(* PLC project 1m8QV2026年3月28日 - 信号稳定延长 - 10ms - 副本.project, CODESYS CODESYS V3.5 SP18 *)
(* stored: creationDateTime 2026-06-03T09:30:15.46669, modificationDateTime 2026-06-01T11:36:08.9259729 *)

(* ============================================================================== DUT: AxisCrtlStruct 作用: 单轴“控制意图”数据结构；每轴各有一份 Local（本控）与 Remote（远控） 使用者: *_Ctrl_FB（读 sCtrl/sLocal）、*_ctrl_1、SecurityCheck、Modbus_Slave ============================================================================== *)
TYPE AxisCrtlStruct : STRUCT
  iMode : INT;  (* 当前请求模式，取值见 MODES 枚举 *)
  rPosCmd : REAL;  (* 位置命令 (deg)，位置/程引模式目标 *)
  rVelCmd : REAL;  (* 速度命令 (deg/s)，速度模式目标 *)
  rPIDCmdVel : LREAL;  (* PID 输出的速度指令（内部，写 CANopen 目标速度前） *)
  rPIDCmdPos : LREAL;  (* PID 目标位置（内部） *)
  bPIDEnable : BOOL;  (* 位置环 PID 使能 *)
  bStartAutoTrack : BOOL;  (* 自跟踪使能：TRUE 时用 rChanU 误差驱动 *)
  rChanU : REAL;  (* 跟踪接收机误差电压（自跟踪通道） *)
  rP : REAL := 1.0;  (* PID 比例系数（正常指向） *)
  rI : REAL := 0;  (* PID 积分系数 *)
  rD : REAL := 0;  (* PID 微分系数 *)
  rPIDThre : INT := 1;  (* 积分开启的位置误差阈值 *)
  rP_AutoTrack : REAL := 3.0;  (* 自跟踪 P *)
  rI_AutoTrack : REAL := 0.02;  (* 自跟踪 I *)
  rAcceleration : REAL := 3;  (* 加速度 (deg/s²)，写 diTargetAcc 前换算 *)
  rDeceleration : REAL := 3;  (* 减速度 (deg/s²) *)
  rJogVel : LREAL := 2;  (* 点动速度 *)
  Pos_Vel : REAL := 4;  (* 位置模式最大趋近速度 (deg/s) *)
  rPos_Limit : LREAL;  (* 位置限位（备用） *)
  rVel_Limit : LREAL := 3;  (* 速度限幅 (deg/s) *)
  rSoft_limit_Postive : REAL;  (* 软限位正限 (deg) *)
  rSoft_limit_Negative : REAL;  (* 软限位负限 (deg) *)
  rLimitionNegative : LREAL;  (* 硬限位负（备用） *)
  rLimitionPositive : LREAL;  (* 硬限位正（备用） *)
END_STRUCT;
END_TYPE

(* ============================================================================== DUT: AxisStatus 作用: 单轴运行状态（由 *_ctrl_1 根据 CANopen 状态字/逻辑填写） 使用者: *_Ctrl_FB（判断 Disabled/Moving）、Modbus 上报、HMI ============================================================================== *)
TYPE AxisStatus : STRUCT
  Valid : BOOL;  (* 轴数据有效（SoftMotion 风格字段，部分逻辑未用） *)
  Busy : BOOL;  (* 轴忙 *)
  Error : BOOL;  (* 有故障（常映射 GVL.bXxxStsBit3） *)
  ErrorID : UINT;  (* 故障码（常映射 eXxxErrorcode） *)
  ErrorStop : BOOL;  (* 故障停机中 *)
  Disabled : BOOL;  (* 伺服未使能/下电状态 *)
  Stopping : BOOL;  (* 正在停止 *)
  Homing : BOOL;  (* 回零中 *)
  Standstill : BOOL;  (* 静止 Standstill *)
  DiscreteMotion : BOOL;  (* 离散运动 *)
  ContinuousMotion : BOOL;  (* 连续运动 *)
  bServo_Enable : BOOL;  (* 伺服已使能（本工程：StsBit0/1/2 均为真） *)
  bBrake : BOOL;  (* 抱闸抱紧（与使能相反） *)
  Moving : BOOL;  (* 是否在运动（ctrl_1 根据速度判断 bStop_x） *)
END_STRUCT;
END_TYPE

(* ============================================================================== DUT: AxisVisible 作用: 本控/HMI 显示与操作相关状态（可视化、按钮灯） 使用者: 可视化或本控面板逻辑（部分工程可能未全部接线） ============================================================================== *)
TYPE AxisVisible : STRUCT
  bJog_Forward : BOOL := FALSE;
  bJog_Backward : BOOL := FALSE;
  bVel_Run : BOOL := FALSE;
  bPos_Run : BOOL := FALSE;
  bEnable : BOOL;  (* 使能指示灯 *)
  bUnable : BOOL;  (* 下使能指示灯 *)
  bLocalCtrl : BOOL;  (* 本控指示灯 *)
  bRemoteCtrl : BOOL;  (* 远控指示灯 *)
  bStop : BOOL;  (* 停止指示灯 *)
  bmoveLight : BOOL;
  bErrLight : BOOL;  (* 报错提示灯 *)
  rLocalPosCmd : REAL;  (* 本控位置命令 *)
  rLocalVelCmd : REAL;  (* 本控速度命令 *)
END_STRUCT;
END_TYPE

(* values of MODES: powerOff: 下电：断开驱动使能、清零控制字; powerOn: 上电：按步序置位 bCtrlBit，准备伺服; positionMode: 位置模式：位置环/指向，远控指向常用; velocityMode: 手动速度模式：直接写目标速度; programBootMode: 程序引导/程引模式：按时间插值位置（RealTimePosCal）; reset: 轴错误复位（配合 GVL.bError_Reset）; halt: 停止：减速停机; stop: 挂机/保持停止; jog: 退限位/点动类模式; edge: 边沿相关模式（工程内扩展用）; test1: 测试/多项式系数下发等扩展模式 *)

(* ============================================================================== DUT: MODES 作用: 三轴运动控制状态机使用的模式枚举（El_Ctrl_FB 等 CASE iMode OF） 用法: sCtrl.iMode / sLocal.iMode 与 MODES.xxx 比较 注意: 数值 5 未使用；test1(11) 用于多项式等特殊调试 ============================================================================== *)
{attribute 'qualified_only'}
{attribute 'strict'}
TYPE MODES : (powerOff := 0, powerOn := 1, positionMode := 2, velocityMode := 3, programBootMode := 4, reset := 6, halt := 7, stop := 8, jog := 9, edge := 10, test1 := 11);
END_TYPE

TYPE Word2Bit : UNION
  Apart_Word : WORD;  (* 整字视图（如 AGC 原始 WORD） *)
  Apart_Byte : ARRAY[1..2] OF BYTE;  (* 按字节拆分，[1][2] 与串口 recBuf 逐字节对接 *)
  Apart_Real : REAL;  (* 按 32 位实数解释（本 UNION 仅 16 位，慎用） *)
  Apart_Int : INT;  (* 有符号整数视图（如 Ua/Ue 误差电压 raw） *)
END_UNION;
END_TYPE

TYPE Dword2Bit : UNION
  Apart_Dword : DWORD;  (* 32 位整字 *)
  Apart_Word : ARRAY[1..2] OF WORD;  (* 拆成两个 16 位寄存器（与 Modbus WORD 对接时常用） *)
  Apart_Byte : ARRAY[1..4] OF BYTE;  (* 4 字节，串口按字节填充 *)
  Apart_Real : REAL;  (* 32 位浮点视图 *)
  Apart_Int : INT;  (* 32 位有符号整数（部分帧解析用 INT） *)
END_UNION;
END_TYPE

TYPE float2bit : UNION
  Apart_ulint : ULINT;  (* 64 位无符号时间戳等 *)
  Apart_dword : ARRAY[1..2] OF DWORD;  (* 两个双字；位置常用 dword[1] 装 DINT *)
  Apart_word : ARRAY[1..4] OF WORD;  (* 四个 Modbus 保持寄存器字 *)
  Apart_byte : ARRAY[1..8] OF BYTE;  (* 8 字节逐字节访问 *)
  Apart_real : ARRAY[1..2] OF REAL;  (* 两个 REAL 视图 *)
  Apart_int : ARRAY[1..4] OF INT;  (* 四个 INT 视图 *)
END_UNION;
END_TYPE

TYPE UnionLREAL_WORD : UNION
  lrealValue : LREAL;  (* 程序内使用的双精度浮点值 *)
  words : ARRAY[1..4] OF WORD;  (* Modbus 4 寄存器拼装/拆分 *)
END_UNION;
END_TYPE

TYPE Time2Word : UNION
  uliData : ULINT;  (* 64 位时间（如 ns/ms 打包，视使用处换算） *)
  wWords : ARRAY[1..4] OF WORD;  (* 与 4 个寄存器对应 *)
  lrReal : LREAL;  (* 双精度时间或系数视图 *)
  arReal : ARRAY[0..1] OF REAL;  (* 两个单精度视图（高低段等） *)
END_UNION;
END_TYPE

PROGRAM PLC_PRG
  VAR
    a : DINT;
    b : REAL;
  END_VAR

                    a := REAL_TO_DINT(b * 524288 / 360);
                  
END_PROGRAM

PROGRAM TimeCase
  VAR
    Triger AT %IX0.0 : BOOL;
    Feed AT %QX0.0 : BOOL;
  END_VAR
  VAR
    stUTC_Timestamp : SYSTIME;
    stSYS_Timestamp : ULINT;
    stGNSS_Timestap : ULINT;
    Result : RTS_IEC_RESULT;
    Uptriger : Standard.R_TRIG;
    TON_F : TON;
    dDelPTime : DINT;
    max_DelPTime : DINT := 0;
    min_DelPTime : DINT := -999999;
    iCount : INT;
    dtNow : DT;
    dtGNSS : DT;
    dtLastGNSS : ULINT;
    iDiffETime : DINT;
    DelPTime : DINT;
  END_VAR

                    //计算时间误差序列
Result := SysTimeRtcHighResGet(stUTC_Timestamp);        
stSYS_Timestamp := TO_ULINT(stUTC_Timestamp);           // ULINT，获取本地时间
dtNow := TO_DT(stUTC_Timestamp / 1000); 		        // 转换为DATE_AND_TIME类型

Uptriger(CLK:=Triger);                                  //检测PPS上升沿
IF Uptriger.Q THEN                                      //上升沿触发后，GPRMC解析，DO0上升沿输出（电平24V）
	Feed:=TRUE;	
	dtGNSS := TO_DT(GVL.stGNSS_Timestap / 1000); 	    // 拿到串口时间数据			                                     
	iDiffETime:=ULINT_TO_DINT(GVL.stGNSS_Timestap-dtLastGNSS);  
	dtLastGNSS:=GVL.stGNSS_Timestap;                    //缓存上一周期时间戳（ms)  
	dDelPTime:=ULINT_TO_DINT(GVL.stGNSS_Timestap - stSYS_Timestamp);       //计算误差	              
	IF iDiffETime = 1000 THEN                           //确保时间更新步进1S
		IF dDelPTime < 0 THEN                           //更新最小值
			IF dDelPTime < min_DelPTime THEN
				min_DelPTime:=dDelPTime;
				DelPTime:=min_DelPTime;                 
			END_IF		
		ELSE                                            //更新最大值
			IF dDelPTime > max_DelPTime THEN
				max_DelPTime:=dDelPTime;
				DelPTime:=max_DelPTime;
			END_IF
		END_IF	
	END_IF				    						
	iCount:=iCount+1;
	IF iCount >= 60 THEN                                //一分钟校一次时间
		GVL.dDelTime:=DelPTime;
		max_DelPTime:=0;
		min_DelPTime:=0;	
		iCount:=0;
	END_IF
	
END_IF
TON_F(IN:=Feed, PT:=T#100MS, Q=>,ET=>);                 //脉宽200ms（测试时延，为了在示波器看波形）
IF TON_F.Q THEN
	Feed:=FALSE;		
END_IF
                  
END_PROGRAM

FUNCTION_BLOCK PID
  VAR_INPUT
    rTarget : REAL;  (* 目标位置 (deg) *)
    rFeedback : REAL;  (* 实际位置反馈 (deg) *)
    rPosLimPositive : LREAL;  (* 软限位正限 (deg)，超出则输出清零 *)
    rPosLimNegative : LREAL;  (* 软限位负限 (deg) *)
    rKp : REAL;  (* 比例系数 *)
    rKi : REAL;  (* 积分系数 *)
    rKd : REAL;  (* 微分系数（当前逻辑未实际使用） *)
    iThreshold : INT;  (* 积分开启阈值 (deg)；-1 = 始终开积分 *)
    bPIDEnable : BOOL;  (* PID 使能，FALSE 时各项清零 *)
    rVelLim : LREAL;  (* 输出速度限幅 (deg/s) *)
  END_VAR
  VAR_OUTPUT
    rPIDOutput : LREAL;  (* PID 输出速度 (deg/s)，写到 diXxTargetVel 前换算 *)
    rPIDtrace : LREAL;  (* 调试/显示用，与 rPIDOutput 相同 *)
  END_VAR
  VAR
    rLastError : LREAL;  (* 上一拍误差（当前版本未使用微分，保留备用） *)
    rErrorNow : LREAL;  (* 当前误差 = rTarget - rFeedback *)
    rIntegralNew : LREAL;  (* 积分累计量 *)
    rDerivativeNew : LREAL;  (* 微分项（未使用） *)
    rDelta : LREAL;  (* 备用 *)
    rProportionNew : LREAL;  (* 比例项 = rErrorNow *)
  END_VAR

                    
(*==============================================================================
  FB: PID（位置环速度输出 PID）
  任务: Canopen 10ms（由 *_Ctrl_FB 调用）
  作用: 输入目标位置与实际位置，输出速度指令（deg/s）
  算法: 比例 + 条件积分（误差小于阈值才累积），无微分
  使用者: El_Ctrl_FB / Az_Ctrl_FB / Ti_Ctrl_FB 中的 VelPID_1/2/3
==============================================================================*)

// ----- 段：PID 使能入口 -----
IF (bPIDEnable>0) THEN //如果PID使能
	IF rTarget=rFeedback THEN
		rPIDOutput:=0;	               // 目标=反馈，输出为 0
	ELSE
	
		rErrorNow:=rTarget-rFeedback;  //计算当前误差 en
		rProportionNew:=rErrorNow;     //比例项

		// ----- 段：条件积分（仅在软限位内、误差小于阈值时才累积）-----
		IF rFeedback>rPosLimNegative AND rFeedback<rPosLimPositive THEN //若在软限位之内，工作时开启积分项
			IF (ABS(rTarget-rFeedback)<iThreshold) THEN//位置差小于积分阈值
				rIntegralNew:= rIntegralNew+rErrorNow; //积分项
			ELSE
				rIntegralNew:=0;
			END_IF;
		ELSE //不在软限位范围内,则积分项为0
			rIntegralNew:=0;
		END_IF

		// ----- 段：PID 求和输出 -----
		rPIDOutPut:=rKp*rProportionNew+rKi*rIntegralNew;
		rPIDtrace:=rKp*rProportionNew+rKi*rIntegralNew;

		// ----- 段：速度限幅（双向） -----
		IF rPIDOutput<(-rVelLim) THEN
			rPIDOutput:=-rVelLim;
		ELSIF rPIDOutput>rVelLim THEN
			rPIDOutput:=rVelLim;
		END_IF
		
		// ----- 段：超软限位时强制输出清零，防止继续向限位方向运动 -----
		IF rFeedback>rPosLimPositive AND rPIDOutput>0 THEN 
			rPIDOutput:=0;
		END_IF
		IF rFeedback<rPosLimNegative AND rPIDOutput<0 THEN
			rPIDOutput:=0;
		END_IF
		
		rLastError:=rErrorNow;//将当前误差赋值给上一次误差
		
	END_IF
ELSE//非使能清零PID各项
	rProportionNew:=0.0;
	rIntegralNew:=0.0;
	rPIDOutput:=0.0;
END_IF





                  
END_FUNCTION_BLOCK

PROGRAM TimeAdd
  VAR
    icount : INT;
    iSecondLast : INT;
  END_VAR

                    
(*==============================================================================
  PRG: TimeAdd（GNSS 秒跳变监测 / 毫秒插值计数）
  任务: Canopen 10ms
  作用:
    - 监测 GPRMC_1.iSecond 是否更新；未更新则 icount 每 10ms +1
    - RealTimePosCal 使用: GVL.dRealTime := GVL.stGNSS_Timestap + 10 * TimeAdd.icount
      即在两次 GNSS 报文之间用 10ms 步进“补时”，保证程引插值时间连续
  说明:
    icount>2000 时清零（约 20s 无新秒则复位，防止溢出跑飞）
==============================================================================*)
// 监测时统串口状态，时间插值
IF iSecondLast <> GPRMC_1.iSecond THEN
	icount := 0;
ELSE
	icount := icount + 1;
END_IF
iSecondLast := GPRMC_1.iSecond;

IF icount > 2000 THEN
	icount := 0;
END_IF
                  
END_PROGRAM

PROGRAM GPRMC
  VAR
    com_init : gcan.FB_Com_Init;  (* gcan.FB_Com_Init为串口初始化功能块，可设定串口端口号，串口波特率等参数 *)
    com_read : gcan.FB_Com_Read;  (* gcan.FB_Com_Read为串口接收功能块，用于通过接收串口发送给PLC的数据 *)
    com_write : gcan.FB_Com_Write;  (* gcan.FB_Com_Write为串口发送功能块，用于发送串口数据 *)
    m_uiError : UINT;  (* 用于承接功能块中报错引脚错误信息的变量 *)
    m_out : BOOL;  (* 用于承接功能块中完成标志引脚数据的变量 *)
    isFirst : BOOL := TRUE;  (* 用于判断初始化只执行一次的逻辑 *)
    mPort : BYTE;  (* 程序中用作设定串口端口号 *)
    recSize : UINT;  (* 接收数据长度，单位：字节 *)
    recBuf : ARRAY[0..100] OF BYTE;  (* 用于存放接收到的串口数据的数组 *)
    sum_i : INT;
    checksum : BYTE;
    iYear : INT;
    iMonth : INT;
    iDay : INT;
    iHour : INT;
    iMinute : INT;
    iSecond : INT;
    strDateTimeNow : STRING;
    gnssTimestamp : ULINT;
    high4 : BYTE;
    low4 : BYTE;
  END_VAR

                    ////////////////////////////////////////////////////////////////////////////////////////
//串口接收GPRMC报文解析
//日期：2024/08/25
//版本：V1.1
/////////////////////////////////////////////////////////////////////////////////////////

mPort:=1;								//串口端口号设定，GCAN-PLC-400、GCAN-PLC-510、GCAN-PLC-511，1为232，2为485
										//GCAN-PLC-324、GCAN-PLC-326，1为第一路485，2为第2路485
IF isFirst THEN
	com_init(							//串口初始化功能块
	EN_IN:=TRUE,						//串口初始化功能块使能
	xEnable:=TRUE,						//串口功能使能
	bPort:=mPort,						//串口端口号设定
	uiBaudrate:=115200,					//串口波特率设定
	bParity:=0,							//串口奇偶校验设定，0为无校验，1为奇校验，2为偶检验
	bDatabits:=8,						//数据位设定
	bStopbits:=1,						//停止位设定
	EN_OUT=>m_out,						//串口初始化功能块执行完成标志位
	uiError=>m_uiError);				//串口初始化功能块执行错误信息
	isfirst:=FALSE;						//执行一次初始化后关闭IF的条件使其之后进入ELSE程序段运行

ELSE
	
		com_read(						//串口读取功能块
		EN_in:=TRUE,					//读取功能块使能，为TRUE执行读取
		bPort:=mPort,					//串口端口号设定
		p_brxdata:=ADR(recBuf),			//读取到的串口数据引脚为指针类型，使用ADR()指向自建数组将数据存放到数组中
		uiMaxsize:=100,					//设定最大读取长度
		EN_out=>m_out,					//串口读取功能块执行完成标志位******功能块执行完成不代表接收完成********
		uiRecSize=>recSize,				//串口接收数据长度，单位：字节，大于0时说明接收到数据可用于判断是否接收
		uierror=>m_uierror);			//串口读取功能块执行错误信息
										//从数组recBuf里取数据，解析出年、月、日、时、分、秒
		//有效判定(A)+和校验(hh),前 4bit和后 4bit的 16 进制数分别以 ASCII 码表示(0~9,A~F)，高位在前。
		IF 	recBuf[17] = 65 THEN
(*			checksum := 16#00;
			FOR sum_i:=1 TO 74 BY 1 DO
				checksum:= checksum XOR recBuf[sum_i];
			END_FOR
			high4 := (SHR(checksum, 4) AND 16#0F)+16#30;
			low4 := (checksum AND 16#0F)+16#30;
			IF recBuf[76]= high4 AND recBuf[77]= low4 THEN 
*)			IF recBuf[60] = 44 THEN // 航向角 x.x
				iYear:=BYTE_TO_INT(recBuf[65]-48)*10+BYTE_TO_INT(recBuf[66]-48)+2000;
				iMonth:=BYTE_TO_INT(recBuf[63]-48)*10+BYTE_TO_INT(recBuf[64]-48);
				iDay:=BYTE_TO_INT(recBuf[61]-48)*10+BYTE_TO_INT(recBuf[62]-48);
				iHour:=BYTE_TO_INT(recBuf[7]-48)*10+BYTE_TO_INT(recBuf[8]-48)+8;
				iMinute:=BYTE_TO_INT(recBuf[9]-48)*10+BYTE_TO_INT(recBuf[10]-48);
				iSecond:=BYTE_TO_INT(recBuf[11]-48)*10+BYTE_TO_INT(recBuf[12]-48);
			END_IF
			IF recBuf[61] = 44 THEN // 航向角 xx.x
				iYear:=BYTE_TO_INT(recBuf[66]-48)*10+BYTE_TO_INT(recBuf[67]-48)+2000;
				iMonth:=BYTE_TO_INT(recBuf[64]-48)*10+BYTE_TO_INT(recBuf[65]-48);
				iDay:=BYTE_TO_INT(recBuf[62]-48)*10+BYTE_TO_INT(recBuf[63]-48);
				iHour:=BYTE_TO_INT(recBuf[7]-48)*10+BYTE_TO_INT(recBuf[8]-48)+8;
				iMinute:=BYTE_TO_INT(recBuf[9]-48)*10+BYTE_TO_INT(recBuf[10]-48);
				iSecond:=BYTE_TO_INT(recBuf[11]-48)*10+BYTE_TO_INT(recBuf[12]-48);
			END_IF
			IF recBuf[62] = 44 THEN // 航向角 xxx.x
				iYear:=BYTE_TO_INT(recBuf[67]-48)*10+BYTE_TO_INT(recBuf[68]-48)+2000;
				iMonth:=BYTE_TO_INT(recBuf[65]-48)*10+BYTE_TO_INT(recBuf[66]-48);
				iDay:=BYTE_TO_INT(recBuf[63]-48)*10+BYTE_TO_INT(recBuf[64]-48);
				iHour:=BYTE_TO_INT(recBuf[7]-48)*10+BYTE_TO_INT(recBuf[8]-48)+8;
				iMinute:=BYTE_TO_INT(recBuf[9]-48)*10+BYTE_TO_INT(recBuf[10]-48);
				iSecond:=BYTE_TO_INT(recBuf[11]-48)*10+BYTE_TO_INT(recBuf[12]-48);
			END_IF
				// 计算时间戳		
				strDateTimeNow := CONCAT(STR1 := 'DT#', STR2 := INT_TO_STRING(iYear));
				strDateTimeNow := CONCAT(STR1 := strDateTimeNow, STR2 := '-');
				strDateTimeNow := CONCAT(STR1 := strDateTimeNow, STR2 := INT_TO_STRING(iMonth));
				strDateTimeNow := CONCAT(STR1 := strDateTimeNow, STR2 := '-');
				strDateTimeNow := CONCAT(STR1 := strDateTimeNow, STR2 := INT_TO_STRING(iDay));
				strDateTimeNow := CONCAT(STR1 := strDateTimeNow, STR2 := '-');
				strDateTimeNow := CONCAT(STR1 := strDateTimeNow, STR2 := INT_TO_STRING(iHour));
				strDateTimeNow := CONCAT(STR1 := strDateTimeNow, STR2 := ':');
				strDateTimeNow := CONCAT(STR1 := strDateTimeNow, STR2 := INT_TO_STRING(iMinute));
				strDateTimeNow := CONCAT(STR1 := strDateTimeNow, STR2 := ':');
				strDateTimeNow := CONCAT(STR1 := strDateTimeNow, STR2 := INT_TO_STRING(iSecond));
				gnssTimestamp := DT_TO_ULINT(TO_DT(strDateTimeNow)) * 1000;
				GVL.stGNSS_Timestap := gnssTimestamp;
			//END_IF
		END_IF
					


(*	IF recsize>0 THEN					//如果接收到串口数据
		
		com_write(						//串口发送功能块
		EN_IN:=TRUE,					//串口发送功能块使能，发送机制：当使能为TRUE时，PLC程序每周期运行到此处就执行一次发送
		bPort:=mPort,					//串口端口号设定
		p_bTxdata:=ADR(recbuf),			//将接收存放到数组中的数据发送出去******若发送其它数据，自建另一数组用于存放发送数据即可
		uiTxsize:=recsize,				//发送长度为接收到的数据长度******若发送其它长度，自行填写所需长度即可
		EN_OUT=>m_out,					//串口发送功能块执行完成标志位
		uierror=>m_uierror);			//串口发送功能块执行错误信息
			
	END_IF
*)	
END_IF
                  
END_PROGRAM

PROGRAM RealTimePosCal
  VAR
    dtReal : DT;
    sRealTime : STRING;
    btestTimeInit : BOOL;
    AzCubicInter : threesimple2_1;  (* 方位三次样条插值 *)
    ElCubicInter : threesimple2_1;  (* 俯仰三次样条插值 *)
    iErrcode : INT;
    rInterAzPos : REAL;  (* 方位轴插值位置 *)
    rInterElPos : REAL;  (* 俯仰轴插值位置 *)
    rInterAzPostest : REAL;  (* 方位轴插值位置 *)
    rInterElPostest : REAL;  (* 俯仰轴插值位置 *)
    rPolyAzPos : REAL;  (* 方位轴多项式位置 *)
    rPolyElPos : REAL;  (* 俯仰轴多项式位置 *)
    AzPoly : Get_AZ;
    ElPoly : Get_AZ_1;
    dRTime : ULINT;  (* 上位机外部时间 单位ns Unix时间戳，起点是1970-1-1 0:0:0 *)
    dLastRTime : ULINT;
    icount : INT;
  END_VAR

                    
(*==============================================================================
  PRG: RealTimePosCal（程引实时位置计算）
  任务: Canopen 10ms
  作用:
    1. 合成 GVL.dRealTime（毫秒时间轴，供插值用 xt）
    2. 双轴程引(mode4)时，按时间对 Modbus 轨道表做三次样条插值
    3. 输出 rInterAzPos / rInterElPos → *_ctrl_1 合成 rPIDCmdPos
  时间源（GVL.bTimeSwich）:
    FALSE — GNSS: stGNSS_Timestap + 10×TimeAdd.icount
    TRUE  — 上位机 UTC: Modbus_Slave.UTC_New + 8h + 10×本地 icount
  插值输入:
    X = Modbus_Slave.aUTC_TIME[1..10]（时间结点，相对首点归一化）
    Y = Modbus_Slave.aPosCmd_1/2（俯仰/方位角度结点）
    xt = dRealTime - 8×3600×1000（转为与轨道表一致的 UTC 毫秒）
==============================================================================*)

// =============================================================================
// 段 1: 合成 GVL.dRealTime（全局毫秒时钟）
// =============================================================================

//直接从上位机拿数（UTC_New 一般为 UTC 毫秒，+8h 对齐北京时）
dRTime := modbus_slave.UTC_New + 8 * 3600 * 1000;
IF dRTime <> dLastRTime THEN
	icount := 0;
ELSE 
	icount := icount + 1;
END_IF
dLastRTime:=dRTime;

IF not GVL.bTimeSwich THEN
	GVL.dRealTime:=GVL.stGNSS_Timestap + 10*timeadd.icount;   // GNSS + 插值
ELSE
	GVL.dRealTime:=dRTime + 10*icount;                        // 上位机 UTC + 插值
END_IF
IF icount > 5000 THEN
	icount := 0;
END_IF
(*
GVL.dRealTime:=GVL.stGNSS_Timestap + 10*timeadd.icount;
*)
dtReal := TO_DT(GVL.dRealTime / 1000);
sRealTime := TO_STRING(dtReal);

// =============================================================================
// 段 2: 双轴均为程引 mode4 时 — 三次样条插值求当前俯仰/方位
// xt 减去 8×3600×1000 与轨道表 aUTC_TIME 时间基准对齐
// =============================================================================
IF Axis1Remote.iMode=4 AND Axis2Remote.iMode=4 THEN//若PTP时间锁定 且时间模式为PTP时间
		//三次样条插值

		//GVL.dRealTime:= TimeCase.stSYS_Timestamp + GVL.dDelTime + 1000 + 56; // 矫正后的时间 单位毫秒
		IF NOT GVL.bTimeSwich THEN
			GVL.dRealTime:=GVL.stGNSS_Timestap + 10*timeadd.icount;
		ELSE
			GVL.dRealTime:=dRTime + 10*icount;
		END_IF
		AzCubicInter(XModbusUL:=Modbus_Slave.aUTC_TIME,YModbus:=Modbus_Slave.aPosCmd_2,y0:=0,yn:=0,xt:=(ULINT_TO_LREAL(GVL.dRealTime) - 8 * 3600 *1000),sout=>rInterAzPos,ErrCode=>iErrcode);
		ElCubicInter(XModbusUL:=Modbus_Slave.aUTC_TIME,YModbus:=Modbus_Slave.aPosCmd_1,y0:=0,yn:=0,xt:=(ULINT_TO_LREAL(GVL.dRealTime) - 8 * 3600 *1000),sout=>rInterElPos,ErrCode=>iErrcode);
		IF iErrcode>0 THEN //模块内错误代码清0 外部维持
			Error_code:=iErrcode;
		END_IF
END_IF

(* 段 3: 多项式拟合程引（Get_AZ / Get_AZ_1）整段已注释，当前未使用
   若启用: rInterAzPos = -rPolyAzPos, rInterElPos = rPolyElPos + 90
*)

                  
END_PROGRAM

PROGRAM Modbus_Slave
  VAR
    modbusData AT %MW0 : ARRAY[0..654] OF WORD;  (* HR 保持寄存器，CODESYS 地址 %MW0 起 *)
    modbusInputRegs AT %MW660 : ARRAY[0..79] OF WORD;  (* IR 输入寄存器，%MW660 起 *)
  END_VAR
  VAR
    modTcpSlaveInit : gcan.FB_ModbusTCP_Slave_Init;  (* ----- Modbus TCP 协议栈 ----- *)
    modTcpSlaveCtrl : gcan.FB_ModbusTCP_Slave_Ctrl;
    eout : BOOL;
    iSocket : INT;
    uiErr : UINT;
    isInit : BOOL;
    arClient : ARRAY[0..10] OF INT;
    arDo_data : ARRAY[0..654] OF BOOL;
    arDi_data : ARRAY[0..79] OF BOOL;
    enCtr : BOOL;
    dif : ULINT;
    iCount : WORD;
    TypeList1 : DWORD;
    UTC_Union : float2bit;  (* HR[0..3] 上位机 UTC 毫秒 *)
    CtrlBool : WORD_AS_BIT;  (* HR[7] 控制字位域 *)
    bCommReset : BOOL;  (* HR[7].14 → SecurityCheck 故障复位 *)
    iWatchDogTime : INT;
    Pos1_Union : float2bit;
    Pos2_Union : float2bit;
    Pos3_Union : float2bit;
    iMode_1 : INT;  (* HR[19] *)
    rPosCmd_1 : REAL;  (* HR[20..21] DINT/1e5 +90° *)
    rVelcmd_1 : REAL;
    rP_1 : REAL;
    rI_1 : REAL;
    rD_1 : REAL;
    rThreshold_1 : INT;
    rAcceleration_1 : REAL;
    rDeceleration_1 : REAL;
    rVelLim_1 : REAL;
    iMode_2 : INT;  (* ----- 方位轴 HR[8..18] ----- *)
    rPosCmd_2 : REAL;  (* ×(-1) 与上报符号约定一致 *)
    rVelcmd_2 : REAL;
    rP_2 : REAL;
    rI_2 : REAL;
    rD_2 : REAL;
    rThreshold_2 : INT;
    rAcceleration_2 : REAL;
    rDeceleration_2 : REAL;
    rVelLim_2 : REAL;
    iMode_3 : INT;
    rPosCmd_3 : REAL;
    rVelcmd_3 : REAL;
    rP_3 : REAL;
    rI_3 : REAL;
    rD_3 : REAL;
    rThreshold_3 : INT;
    rAcceleration_3 : REAL;
    rDeceleration_3 : REAL;
    rVelLim_3 : REAL;
    UTC_Orbit_Union : float2bit;
    UTC_Orbit_New : ULINT;
    UTC_Orbit_Last : ULINT;
    TimeBias_Union : float2bit;
    Bias1_Union : float2bit;
    Bias2_Union : float2bit;
    Bias3_Union : float2bit;
    AcuElOffset : float2bit;
    rTimeBias : LREAL;
    rBias_1 : LREAL;
    rBias_2 : LREAL;
    rBias_3 : LREAL;
    lrElOffset : LREAL;
    UTC_New : ULINT;
    UTC_Last : ULINT;
    aUTC_TIME : ARRAY[1..10] OF ULINT;  (* ----- 程引轨道表（10 点时间与角度序列）→ RealTimePosCal 插值 ----- *)
    aPosCmd_1 : ARRAY[1..10] OF LREAL;  (* 俯仰 *)
    aPosCmd_2 : ARRAY[1..10] OF LREAL;  (* 方位 *)
    isave : INT;
    iCheck : INT;
    bPass : BOOL;
    iclear : INT;
    uPTPTime_Union : float2bit;
    DI1_Union : Util.BIT_AS_WORD;
    DI2_Union : Util.BIT_AS_WORD;
    DO1_Union : Util.BIT_AS_WORD;
    DO2_Union : Util.BIT_AS_WORD;
    DI1_word : WORD;
    DI2_word : WORD;
    DO1_word : WORD;
    DO2_word : WORD;
    PosSub1_Union : float2bit;
    PosSub2_Union : float2bit;
    PosSub3_Union : float2bit;
    BiasSub1_Union : float2bit;
    BiasSub2_Union : float2bit;
    BiasSub3_Union : float2bit;
    Chan_Union : Util.BIT_AS_WORD;
    Chan_word : WORD;
    ptptime : ULINT;
    rAzTheory : LREAL;
    rEltheory : LREAL;
    rAzTheory_Union : float2bit;
    rEltheory_Union : float2bit;
    MillisecondsTime : ULINT;
    DeltaTimeBetPC : ULINT;
    AGC_Value : REAL;
    starttime : LREAL;
    rNodeTime1_az : LREAL;
    rNodeTime2_az : LREAL;
    rNodeTime3_az : LREAL;
    rNodeTime4_az : LREAL;
    rNodeTime5_az : LREAL;
    rEndTime : LREAL;
    lrFun1_az : ARRAY[0..10] OF LREAL;
    lrFun2_az : ARRAY[0..10] OF LREAL;
    lrFun3_az : ARRAY[0..10] OF LREAL;
    lrFun4_az : ARRAY[0..10] OF LREAL;
    lrFun5_az : ARRAY[0..10] OF LREAL;
    lrFun6_az : ARRAY[0..10] OF LREAL;
    unionFun1_az : ARRAY[0..10] OF UnionLREAL_WORD;
    unionFun2_az : ARRAY[0..10] OF UnionLREAL_WORD;
    unionFun3_az : ARRAY[0..10] OF UnionLREAL_WORD;
    unionFun4_az : ARRAY[0..10] OF UnionLREAL_WORD;
    unionFun5_az : ARRAY[0..10] OF UnionLREAL_WORD;
    unionFun6_az : ARRAY[0..10] OF UnionLREAL_WORD;
    unionStartTime : UnionLREAL_WORD;
    unionNodeTime1_az : UnionLREAL_WORD;
    unionNodeTime2_az : UnionLREAL_WORD;
    unionNodeTime3_az : UnionLREAL_WORD;
    unionNodeTime4_az : UnionLREAL_WORD;
    unionNodeTime5_az : UnionLREAL_WORD;
    unionEndTime : UnionLREAL_WORD;
    rNodeTime1_el : REAL;
    rNodeTime2_el : REAL;
    rNodeTime3_el : REAL;
    rNodeTime4_el : REAL;
    rNodeTime5_el : REAL;
    lrFun1_el : ARRAY[0..10] OF LREAL;
    lrFun2_el : ARRAY[0..10] OF LREAL;
    lrFun3_el : ARRAY[0..10] OF LREAL;
    lrFun4_el : ARRAY[0..10] OF LREAL;
    lrFun5_el : ARRAY[0..10] OF LREAL;
    lrFun6_el : ARRAY[0..10] OF LREAL;
    unionFun1_el : ARRAY[0..10] OF UnionLREAL_WORD;
    unionFun2_el : ARRAY[0..10] OF UnionLREAL_WORD;
    unionFun3_el : ARRAY[0..10] OF UnionLREAL_WORD;
    unionFun4_el : ARRAY[0..10] OF UnionLREAL_WORD;
    unionFun5_el : ARRAY[0..10] OF UnionLREAL_WORD;
    unionFun6_el : ARRAY[0..10] OF UnionLREAL_WORD;
    unionNodeTime1_el : UnionLREAL_WORD;
    unionNodeTime2_el : UnionLREAL_WORD;
    unionNodeTime3_el : UnionLREAL_WORD;
    unionNodeTime4_el : UnionLREAL_WORD;
    unionNodeTime5_el : UnionLREAL_WORD;
    unionSum : UnionLREAL_WORD;
    lrSum : LREAL;
    lrSumlocal : LREAL;
    i : INT;
    bNotFirst : BOOL;
    bCheck : BOOL;
    bIFPoly : BOOL;
    iCountPolyGet : INT;
    uChangeTest : Time2Word;
    iCountSum : INT;
    bSearch : BOOL;  (* HR[7].6 十字/AGC 搜索 *)
    bStartTrackAcu : BOOL;  (* HR[7].10 ACU 请求自跟踪 *)
    rAzPosVel : REAL;
    rElPosVel : REAL;
    rTlPosVel : REAL;
  END_VAR

                    (*==============================================================================
  PRG: Modbus_Slave（Modbus TCP 从站网关）
  任务: MainTask 50ms
  协议: Modbus TCP 端口 502，GCAN FB_ModbusTCP_Slave_*

  内存映射（与 GVL AT %MW 一致）:
    modbusData      AT %MW0   — 保持寄存器 HR，上位机读写（下发命令+多项式系数）
    modbusInputRegs AT %MW660 — 输入寄存器 IR，PLC 写入、上位机只读（状态上报）

  数据流:
    上位机写 HR → 本程序解析 → iMode_x/rPosCmd_x/aUTC_TIME 等
                              → SecurityCheck 写 AxisXRemote
    PLC 状态 → 打包 IR → 上位机读

  扩展自定义寄存器: 在 HR 区 modbusData[n] 增加解析/在 IR 区赋值即可
==============================================================================*)
// =============================================================================
// 段 A: Modbus TCP 从站初始化（端口 502，仅首次）
// =============================================================================
IF isInit=FALSE THEN							
	
	modtcpslaveinit(en_in:=TRUE,					//Modbus TCP Slave初始化功能块使能
	xenable:=TRUE,									//使能初始化功能
	iport:=502,										//开放端口号502
	en_out=>eout,									//Modbus TCP Slave初始化功能块执行完成
	isocket=>iSocket,								//创建的socket存入变量
	uierror=>uiErr);								//Modbus TCP Slave初始化功能块执行错误信息
	
	IF isocket>=0 AND uiErr=0 THEN					//成功创建socket且无错误，逻辑标志置位，下周期执行ELSE
		isInit:=TRUE;	
		
		enCtr:=FALSE;
		ELSE                                        //等待连接成功
		modtcpslaveinit(en_in:=0,xenable:=0);	
	END_IF
	
 
ELSE

// =============================================================================
// 段 B: 从站周期服务 — 映射 HR/IR 缓冲区，看门狗 2000ms
// =============================================================================
	modtcpslavectrl(en_in:=enCtr,					//Modbus TCP Slave执行功能块使能
	xenable:=TRUE,									//Modbus TCP Slave执行功能使能
	isocket:=isocket,								//输入创建的socket
	dwatchdogtime:=2000,							//看门狗时间
	p_clientsocket:=ADR(arClient),					//将连接进来的socket存放到数组
	imaxclientcount:=10,							//设置最大连接数量
	uido_number:=10,uido_startaddr:=0,pdo_data:=ADR(ardo_data),		//uido_number设定线圈个数，uido_startaddr设定线圈起始地址，数据存放在ardo_data数组
	uidi_number:=10,uidi_startaddr:=0,pdi_data:=ADR(ardi_data),		//uidi_number设定离散型数据个数，uidi_startaddr设定离散型数据起始地址，数据存放在ardi_data数组
	uireg_number:=655,uireg_startaddr:=0,preg_data:=ADR(modbusData), //uireg_number设定保持型寄存器个数，uireg_startaddr设定保持型寄存器起始地址，数据存放在arreg_data数组
	uiai_number:=79,uiai_startaddr:=0,pai_data:=ADR(modbusInputRegs),//uiai_number设定输入型寄存器个数，uiai_startaddr设定输入型寄存器起始地址，数据存放在arai_data数组
	en_out=>eout,									//Modbus TCP Slave执行功能块执行完成
	uierror=>uierr);								//Modbus TCP Slave执行功能块执行错误信息
	enctr:=TRUE;
	IF uierr <>0 THEN                               //如果从站报错，则重新连接从站
		modtcpslaveinit(en_in:=0,xenable:=0);	
		isInit:=0;
	END_IF
	//iMode:  0 下电  1 上电  2 速度模式  3 停止  4 位置模式  5 继续运行
	//方位轴指令
(*
	Az_ctrl.iMode:=WORD_TO_INT(modbusData[0]);
	AZ_ctrl.rTarVel:=WORD_TO_REAL(modbusData[1]);
	AZ_ctrl.rTarPos:=WORD_TO_REAL(modbusData[2])*-1.0;
	
	//俯仰轴指令
	El_ctrl.iMode:=WORD_TO_INT(modbusData[10]);
	El_ctrl.rTarVel:=WORD_TO_REAL(modbusData[11]);
	El_ctrl.rTarPos:=WORD_TO_REAL(modbusData[12])+90.0;
	*)
	
	// =============================================================================
	// 段 C: 解析 HR 下发（保持寄存器 modbusData → 内部变量）
	// HR[0..3] UTC  HR[7] 控制字  HR[8..18]Az  HR[19..29]El  HR[30..39]Ti
	// HR[43] AGC门限  HR[45..48]轨道时间  HR[51..54]拉偏  HR[57..58]俯仰零位
	// =============================================================================
	UTC_Union.Apart_word[1]:=modbusData[3];
	UTC_Union.Apart_word[2]:=modbusData[2];
	UTC_Union.Apart_word[3]:=modbusData[1];
	UTC_Union.Apart_word[4]:=modbusData[0];
	UTC_New:=UTC_Union.Apart_ulint;
	DeltaTimeBetPC := UTC_New - TO_ULINT(GVL.dRealTime);
	// HR[7] 控制字位定义（WORD_AS_BIT）
	CtrlBool(W:=modbusData[7],
			B14=>bCommReset,
			B13=>Axis2Remote.bPIDEnable,
			B12=>Axis1Remote.bPIDEnable,
			B11=>Axis3Remote.bPIDEnable,
			B10=>bStartTrackAcu,
			B07=>bIFPoly,
			B06=>bSearch, //十字搜索开启标识
			);
	//方位轴指令
	iMode_2:=WORD_TO_INT(modbusData[8]);
	Pos2_Union.Apart_word[2]:=modbusData[9];
	Pos2_Union.Apart_word[1]:=modbusData[10];
	rPosCmd_2:=DINT_TO_LREAL( DWORD_TO_DINT( Pos2_Union.Apart_dword[1]))/100000*-1;
	rVelcmd_2:=DINT_TO_LREAL( WORD_TO_INT(modbusData[11]))/1000*-1;
	rP_2:=INT_TO_LREAL(WORD_TO_INT(modbusData[12]))/1000;
	rI_2:=INT_TO_LREAL(WORD_TO_INT(modbusData[13]))/1000;
	rD_2:=INT_TO_LREAL(WORD_TO_INT(modbusData[14]))/1000;
	rThreshold_2:=WORD_TO_INT(modbusData[15])/1000;
	rAcceleration_2:=INT_TO_LREAL(WORD_TO_INT(modbusData[16]))/1000;
	rDeceleration_2:=INT_TO_LREAL(WORD_TO_INT(modbusData[17]))/1000;
	rVelLim_2:=INT_TO_LREAL(WORD_TO_INT(modbusData[18]))/1000;
	
	//俯仰轴指令
	iMode_1:=WORD_TO_INT(modbusData[19]);
	Pos1_Union.Apart_word[2]:=modbusData[20];
	Pos1_Union.Apart_word[1]:=modbusData[21];
	rPosCmd_1:=DINT_TO_LREAL( DWORD_TO_DINT( Pos1_Union.Apart_dword[1]))/100000+90;
	rVelcmd_1:=DINT_TO_LREAL( WORD_TO_INT(modbusData[22]))/1000;
	rP_1:=INT_TO_LREAL(WORD_TO_INT(modbusData[23]))/1000;
	rI_1:=INT_TO_LREAL(WORD_TO_INT(modbusData[24]))/1000;
	rD_1:=INT_TO_LREAL(WORD_TO_INT(modbusData[25]))/1000;
	rThreshold_1:=WORD_TO_INT(modbusData[26])/1000;
	rAcceleration_1:=INT_TO_LREAL(WORD_TO_INT(modbusData[27]))/1000;
	rDeceleration_1:=INT_TO_LREAL(WORD_TO_INT(modbusData[28]))/1000;
	rVelLim_1:=INT_TO_LREAL(WORD_TO_INT(modbusData[29]))/1000;
	
	//倾斜轴指令
	iMode_3:=WORD_TO_INT(modbusData[30]);
	Pos3_Union.Apart_word[2]:=modbusData[31];
	Pos3_Union.Apart_word[1]:=modbusData[32];
	rPosCmd_3:=DINT_TO_LREAL( DWORD_TO_DINT( Pos3_Union.Apart_dword[1]))/100000*-1;
	rVelcmd_3:=DINT_TO_LREAL( WORD_TO_INT(modbusData[33]))/1000*-1;
	rP_3:=INT_TO_LREAL(WORD_TO_INT(modbusData[34]))/1000;
	rI_3:=INT_TO_LREAL(WORD_TO_INT(modbusData[35]))/1000;
	rD_3:=INT_TO_LREAL(WORD_TO_INT(modbusData[36]))/1000;
	rThreshold_3:=WORD_TO_INT(modbusData[37])/1000;
	rAcceleration_3:=INT_TO_LREAL(WORD_TO_INT(modbusData[38]))/1000;
	rDeceleration_3:=INT_TO_LREAL(WORD_TO_INT(modbusData[39]))/1000;
	
	
	//AGC锁定门限
	AGC_Value:=(WORD_TO_UDINT(modbusData[43])/100.0);
	GVL.Chanthreshold:=AGC_Value;
	
	//轨道时间
	UTC_Orbit_Union.Apart_word[1]:=modbusData[48];
	UTC_Orbit_Union.Apart_word[2]:=modbusData[47];
	UTC_Orbit_Union.Apart_word[3]:=modbusData[46];
	UTC_Orbit_Union.Apart_word[4]:=modbusData[45];
	UTC_Orbit_New:=UTC_Orbit_Union.Apart_ulint;
	//时间拉偏
	TimeBias_Union.Apart_word[1]:=modbusData[50];
	TimeBias_Union.Apart_word[2]:=modbusData[49];
	rTimeBias:=DINT_TO_LREAL( DWORD_TO_DINT( TimeBias_Union.Apart_dword[1]))/100000.0; //单位为秒
	IF rTimeBias>0.4 THEN//时间偏置最大限制 正负0.4秒
		rTimeBias:=0.4;
	ELSIF rTimeBias<-0.4 THEN
		rTimeBias:=-0.4;
	END_IF
	rTimeBias:=rTimeBias*1000000000;//秒转纳秒
	//两轴拉偏
	Bias2_Union.Apart_word[1]:=modbusData[52];
	Bias2_Union.Apart_word[2]:=modbusData[51];
	rBias_2:=DINT_TO_LREAL( DWORD_TO_DINT( Bias2_Union.Apart_dword[1]))/100000.0*(-1);
	
	Bias1_Union.Apart_word[1]:=modbusData[54];
	Bias1_Union.Apart_word[2]:=modbusData[53];
	rBias_1:=DINT_TO_LREAL( DWORD_TO_DINT( Bias1_Union.Apart_dword[1]))/100000.0;
	
	//俯仰零值
	AcuElOffset.Apart_word[1]:=modbusData[58];
	AcuElOffset.Apart_word[2]:=modbusData[57];
	lrElOffset:=DINT_TO_LREAL( DWORD_TO_DINT( AcuElOffset.Apart_dword[1]))/100000.0;
	// ----- 程引轨道表: UTC_Orbit_New 递增时移位写入 aUTC_TIME / aPosCmd_x -----
	
	// 指向模式最大速度 HR[61..63] → GVL.AxisXRemote.Pos_Vel
	rAzPosVel:=INT_TO_LREAL(WORD_TO_INT(modbusData[61]))/1000.0;
	rElPosVel:=INT_TO_LREAL(WORD_TO_INT(modbusData[62]))/1000.0;
	rTlPosVel:=INT_TO_LREAL(WORD_TO_INT(modbusData[63]))/1000.0;
	
	IF rAzPosVel <= 16.0 THEN
		GVL.Axis2Remote.Pos_Vel := rAzPosVel;
	ELSE
		GVL.Axis2Remote.Pos_Vel := 16;
	END_IF
	
	IF rElPosVel <= 11.0 THEN
		GVL.Axis1Remote.Pos_Vel := rElPosVel;
	ELSE
		GVL.Axis1Remote.Pos_Vel := 11;
	END_IF
	
	IF rTlPosVel <= 8.0 THEN
		GVL.Axis3Remote.Pos_Vel := rTlPosVel;
	ELSE
		GVL.Axis3Remote.Pos_Vel := 8;
	END_IF
	
	FOR iCheck:=1 TO 10 DO
		IF UTC_Orbit_New>aUTC_TIME[iCheck] THEN
			bPass:=TRUE;
		ELSE
			bPass:=FALSE;
			EXIT;
		END_IF
	END_FOR
	IF bPass THEN //命令刷新，则更新序列
		FOR isave:=1 TO 9 DO
			aUTC_TIME[isave]:=aUTC_TIME[isave+1];
			aPosCmd_1[isave]:=aPosCmd_1[isave+1];
			aPosCmd_2[isave]:=aPosCmd_2[isave+1];
		END_FOR
		aUTC_TIME[10]:=UTC_Orbit_New;
		aPosCmd_1[10]:=rPosCmd_1;
		aPosCmd_2[10]:=rPosCmd_2;
	END_IF
	//若不是程引模式，则清空轨道时间数据
	IF Axis1Remote.iMode<>4 AND Axis2Remote.iMode<>4 THEN
		FOR iCheck:=1 TO 10 DO
			aUTC_TIME[iCheck]:=0;;
		END_FOR
	END_IF
	
	// =============================================================================
	// 段 D: 打包 IR 上报（modbusInputRegs，上位机只读）
	// IR[0..3]时间 IR[5]Error IR[6..9]DI/DO IR[10+]三轴状态 IR[59..65]跟踪机
	// IR[69..74]跟踪偏差 IR[75..78]理论角
	// =============================================================================
	IF icount<16#FFFF THEN
		icount:=icount+1;
	ELSE
		icount:=0;
	END_IF
	
	DI1_Union(B15:=SecurityCheck.bPrelimit_Positive_1,						//俯仰轴预限位--正 B15=0为未触发，B15=1为触发
			B14:=SecurityCheck.bFinallimit_1,								//俯仰轴终限位
			B13:=SecurityCheck.bPrelimit_Negative_1,						//俯仰轴预限位--负
			B12:=SecurityCheck.bFinallimit_1,								//俯仰位终限位
			B11:=SecurityCheck.bPrelimit_Positive_2,						//方位轴预限位--正
			B10:=SecurityCheck.bFinallimit_2,								//方位轴终限位
			B09:=SecurityCheck.bPrelimit_Negative_2,						//方位轴预限位--负
			B08:=SecurityCheck.bFinallimit_2,								//方位轴终限位
			B07:=FALSE,												//倾斜预限位--正
			B06:=FALSE,												//倾斜终限位--正
			B05:=FALSE,												//倾斜预限位--负
			B04:=FALSE,												//倾斜终限位--负
			B03:=FALSE,												//方位轴过零检测
			B02:=Axis2Status.bBrake,								//方位轴抱闸状态 0为解抱闸，1为抱闸
			B01:=Axis1Status.bBrake,								//俯仰轴抱闸状态
			B00:=Axis3Status.bBrake,								//倾斜轴抱闸状态
			W=>DI1_word	);
			
	DI2_Union(B15:=FALSE,								//
			B14:=FALSE,								//
			B13:=FALSE,
			B12:=FALSE,
			B11:=FALSE,
			B10:=FALSE,
			B09:=FALSE,
			B08:=FALSE,
			B07:=FALSE,
			B06:=FALSE,
			B05:=GVL.bError_Reset,											//错误复位符
			B04:=GVL.bLocalCtrl,											//本远控标识符
			B03:=FALSE,									//退限位标识符
			B02:=Axis2Remote.bPIDEnable,											//方位轴PID使能状态
			B01:=Axis1Remote.bPIDEnable,											//俯仰轴PID使能状态
			B00:=Axis3Remote.bPIDEnable,											//倾斜轴PID使能状态
			W=>DI2_word);
	DO1_Union(B15:=FALSE,								//中心体急停指示灯
			B14:=FALSE,							//声光报警		1为触发，0为未触发
			B13:=FALSE,							//爬梯急停指示灯 B13=1为亮 B13=0为灭
			B12:=FALSE,							//机柜蜂鸣器	B12=1为触发，B12=0为未触发
			B11:=FALSE,							//限位释放指示灯 同上 
			B10:=FALSE,						//本远控指示灯	B10=1为本控，B10=0为远控
			B09:=FALSE,							//系统状态指示灯 B09=1为异常，B09=0为正常	
			B08:=Axis2Status.bBrake,								//方位轴抱闸输出 B08=1为抱闸输出 B08=1为解抱闸输出
			B07:=Axis1Status.bBrake,								//俯仰轴抱闸输出 同上
			B06:=Axis3Status.bBrake,								//倾斜轴抱闸输出 同上
			B05:=FALSE,										//方位风扇输出	B05=1为风扇运行，B05=0为风扇未运行
			B04:=FALSE,										//俯仰风扇输出	同上
			B03:=FALSE,										//倾斜风扇输出	同上
			B02:=Axis2Status.bServo_Enable,									//方位轴供电
			B01:=Axis1Status.bServo_Enable,									//俯仰轴供电
			B00:=Axis3Status.bServo_Enable,									//倾斜轴供电
			W=>DO1_word);
	DO2_Union(B15:=Axis2Status.bServo_Enable,//NOT(Axis1Status.Disabled),						//方位主电机使能状态
			B14:=Axis2Status.bServo_Enable,//NOT(Axis1Status.Disabled),							//方位从电机使能状态
			B13:=Axis1Status.bServo_Enable,//NOT(Axis2Status.Disabled),							//俯仰主电机使能状态		
			B12:=Axis1Status.bServo_Enable,//NOT(Axis2Status.Disabled),							//俯仰从电机使能状态
			B11:=Axis3Status.bServo_Enable,		//倾斜主电机使能状态
	 		B10:=Axis3Status.bServo_Enable,		//倾斜从电机使能状态
			B09:=Az_ctrl_1.bStop_2,			//方位轴主电机停止标识符
	 		B08:=Az_ctrl_1.bStop_2,					  //方位轴从电机停止标识符
	 		B07:=El_ctrl_1.bStop_1,		    //俯仰轴主电机停止标识符
			B06:=El_ctrl_1.bStop_1,				//俯仰轴从电机停止标识符
	 		B05:=Ti_ctrl_1.bStop_3,							//倾斜轴主电机停止标识符
			B04:=Ti_ctrl_1.bStop_3,							//倾斜轴从电机停止标识符
	 		B03:=0,
	 		B02:=0,
			B01:=0,
			B00:=0,
			W=>DO2_word	);
	
	//命令角与实际角偏差
	IF bLocalCtrl THEN
		IF  Axis1Local.iMode=4 THEN
			BiasSub1_Union.Apart_dword[1]:=DINT_TO_DWORD( REAL_TO_DINT((Axis1Local.rPosCmd-rFctPosReal_1)*100000.0));//读取位置
		ELSE
			BiasSub1_Union.Apart_dword[1]:=0;//读取位置
		END_IF
	ELSE
		IF Axis1Remote.iMode=2  THEN 
			BiasSub1_Union.Apart_dword[1]:=DINT_TO_DWORD( REAL_TO_DINT((Axis1Remote.rPosCmd-rFctPosReal_1)*100000.0));//读取位置
		ELSIF Axis1Remote.iMode=4 THEN
			BiasSub1_Union.Apart_dword[1]:=DINT_TO_DWORD( REAL_TO_DINT((RealTimePosCal.rInterElPos-rFctPosReal_1)*100000.0));//读取位置
		ELSE
			BiasSub1_Union.Apart_dword[1]:=0;//读取位置
		END_IF
	END_IF
	
	IF bLocalCtrl THEN
		IF Axis2Local.iMode=4 THEN
			BiasSub2_Union.Apart_dword[1]:=DINT_TO_DWORD( REAL_TO_DINT((Axis2Local.rPosCmd-rFctPosReal_2)*100000.0));//读取位置
		ELSE
			BiasSub2_Union.Apart_dword[1]:=0;//读取位置
		END_IF
	ELSE
		IF Axis2Remote.iMode=2 THEN
			BiasSub2_Union.Apart_dword[1]:=DINT_TO_DWORD( REAL_TO_DINT((Axis2Remote.rPosCmd-rFctPosReal_2)*100000.0));//读取位置
		ELSIF Axis2Remote.iMode=4 THEN
			BiasSub2_Union.Apart_dword[1]:=DINT_TO_DWORD( REAL_TO_DINT((rFctPosReal_2-RealTimePosCal.rInterAzPos)*100000.0));//读取位置
		ELSE
			BiasSub2_Union.Apart_dword[1]:=0;//读取位置
		END_IF
	END_IF
	
	IF bLocalCtrl THEN
		IF Axis3Local.iMode=4 THEN
			BiasSub3_Union.Apart_dword[1]:=DINT_TO_DWORD( REAL_TO_DINT((Axis3Local.rPosCmd-rFctPosReal_3)*100000.0));//读取位置
		ELSE
			BiasSub3_Union.Apart_dword[1]:=0;//读取位置
		END_IF
	ELSE
		IF Axis3Remote.iMode=2 THEN
			BiasSub3_Union.Apart_dword[1]:=DINT_TO_DWORD( REAL_TO_DINT((Axis3Remote.rPosCmd-rFctPosReal_3)*100000.0));//读取位置
		ELSIF Axis2Remote.iMode=4 THEN
			BiasSub3_Union.Apart_dword[1]:=DINT_TO_DWORD( REAL_TO_DINT((Axis3Remote.rPIDCmdPos-rFctPosReal_3)*100000.0));//读取位置
		ELSE
			BiasSub3_Union.Apart_dword[1]:=0;//读取位置
		END_IF
	END_IF
	
	// uPTPTime_Union.Apart_ulint:=TO_ULINT(GVL.dPTPCSTTime/1000000);
	uPTPTime_Union.Apart_ulint:=TO_ULINT((GVL.dRealTime - 8 * 3600 * 1000) * 1000000);
	modbusInputRegs[0]:=uPTPTime_Union.Apart_word[4];
	modbusInputRegs[1]:=uPTPTime_Union.Apart_word[3];
	modbusInputRegs[2]:=uPTPTime_Union.Apart_word[2];
	modbusInputRegs[3]:=uPTPTime_Union.Apart_word[1];
	modbusInputRegs[4]:=INT_TO_WORD( icount);
	modbusInputRegs[5]:=INT_TO_WORD(Error_code);//错误代码
	modbusInputRegs[6]:=DI1_word;
	modbusInputRegs[7]:=DI2_word;
	modbusInputRegs[8]:=DO1_word;
	modbusInputRegs[9]:=DO2_word;
	
	
	PosSub1_Union.Apart_dword[1]:=DINT_TO_DWORD( REAL_TO_DINT((rFctPosReal_1-90)*100000.0));//读取俯仰位置
	
	PosSub2_Union.Apart_dword[1]:=DINT_TO_DWORD( REAL_TO_DINT((rFctPosReal_2*-1)*100000.0));//读取方位位置
	
	PosSub3_Union.Apart_dword[1]:=DINT_TO_DWORD( REAL_TO_DINT((rFctPosReal_3*-1)*100000.0));//读取倾斜位置
	
	
	//方位轴状态
	modbusInputRegs[10]:=INT_TO_WORD(Axis2Remote.iMode);
	
	modbusInputRegs[13]:=PosSub2_Union.Apart_word[2];
	modbusInputRegs[14]:=PosSub2_Union.Apart_word[1];
	
	modbusInputRegs[17]:=INT_TO_WORD(REAL_TO_INT(rFctVelReal_2*1000.0));							//速度
	
	modbusInputRegs[19]:=REAL_TO_UINT(Axis2Remote.rP*1000);
	modbusInputRegs[20]:=REAL_TO_UINT(Axis2Remote.rI*1000);
	modbusInputRegs[21]:=REAL_TO_UINT(Axis2Remote.rD*1000);
	modbusInputRegs[22]:=REAL_TO_UINT(Axis2Remote.rPIDThre*1000);
	modbusInputRegs[23]:=INT_TO_WORD(REAL_TO_INT(securitycheck.rAzCurrent*100.0));
	
	
	//俯仰轴状态
	modbusInputRegs[27]:=INT_TO_WORD(Axis1Remote.iMode);
	
	modbusInputRegs[30]:=PosSub1_Union.Apart_word[2];
	modbusInputRegs[31]:=PosSub1_Union.Apart_word[1];
	
	modbusInputRegs[34]:=INT_TO_WORD(REAL_TO_INT(rFctVelReal_1*1000));							     //速度
	
	modbusInputRegs[36]:=REAL_TO_UINT(Axis1Remote.rP*1000);
	modbusInputRegs[37]:=REAL_TO_UINT(Axis1Remote.rI*1000);
	modbusInputRegs[38]:=REAL_TO_UINT(Axis1Remote.rD*1000);
	modbusInputRegs[39]:=REAL_TO_UINT(Axis1Remote.rPIDThre*1000);
	modbusInputRegs[40]:=INT_TO_WORD(REAL_TO_INT(securitycheck.rElCurrent*100.0));
	//倾斜轴状态
	modbusInputRegs[44]:=INT_TO_WORD(Axis3Remote.iMode);
	
	modbusInputRegs[47]:=PosSub3_Union.Apart_word[2];
	modbusInputRegs[48]:=PosSub3_Union.Apart_word[1];
	
	modbusInputRegs[51]:=INT_TO_WORD(REAL_TO_INT(rFctVelReal_3*1000.0));							//速度
	
	modbusInputRegs[53]:=REAL_TO_UINT(Axis3Remote.rP*1000);
	modbusInputRegs[54]:=REAL_TO_UINT(Axis3Remote.rI*1000);
	modbusInputRegs[55]:=REAL_TO_UINT(Axis3Remote.rD*1000);
	modbusInputRegs[56]:=REAL_TO_UINT(Axis3Remote.rPIDThre*1000);
	modbusInputRegs[57]:=INT_TO_WORD(REAL_TO_INT(securitycheck.rTlCurrent*100.0));
	//跟踪接收机预留
	
	modbusInputRegs[69]:=BiasSub2_Union.Apart_word[2];
	modbusInputRegs[70]:=BiasSub2_Union.Apart_word[1];
	modbusInputRegs[71]:=BiasSub1_Union.Apart_word[2];
	modbusInputRegs[72]:=BiasSub1_Union.Apart_word[1];
	modbusInputRegs[73]:=BiasSub3_Union.Apart_word[2];
	modbusInputRegs[74]:=BiasSub3_Union.Apart_word[1];
	//上报用于校相的方位俯仰轴理论值 （插值位置加当前拉偏位置）
	rAzTheory:=RealTimePosCal.rInterAzPos*(-1);
	rAzTheory_Union.Apart_dword[1]:=DINT_TO_DWORD(LREAL_TO_DINT(rAzTheory*100000.0));
	rEltheory:=RealTimePosCal.rInterElPos-90;
	rEltheory_Union.Apart_dword[1]:=DINT_TO_DWORD(LREAL_TO_DINT(rEltheory*100000.0));
	modbusInputRegs[75]:=rAzTheory_Union.Apart_word[2];
	modbusInputRegs[76]:=rAzTheory_Union.Apart_word[1];
	modbusInputRegs[77]:=rEltheory_Union.Apart_word[2];
	modbusInputRegs[78]:=rEltheory_Union.Apart_word[1];

	//跟踪接收机状态字上报
	Chan_Union(B15:=GVL.Chan1Lock,
			  B14:=GVL.Chan1Online,
			  B13:=GVL.Chan2Lock,
			  B12:=GVL.Chan2Online,
			  //B11:=GVL.bStartTrack,
			  B11:=Read_485.bEBN0Lock,
			  B10:=0,
			  B09:=0,
			  B08:=0,
			  B07:=0,
			  B06:=0,
			  B05:=0,
			  B04:=0,
			  B03:=0,
			  B02:=0,
			  B01:=0,
			  B00:=0,
			  w=>Chan_word);
			  (*
	IF GVL.Chan1AGC >= GVL.Chanthreshold THEN
		GVL.Chan1Lock:=TRUE;
	ELSE
		GVL.Chan1Lock:=FALSE;	
	END_IF
	*)
	//跟踪接收机数据上报
	// IF Ether_Cat.EL6022State=8 THEN
	IF TRUE THEN
			modbusInputRegs[59]:=Chan_word;
			modbusInputRegs[60]:=REAL_TO_WORD(GVL.Chan1AGC*1000);
			
	   IF GVL.Chan1Ua>0 THEN
			modbusInputRegs[61]:=REAL_TO_WORD(GVL.Chan1Ua*1000);
	   ELSE
			modbusInputRegs[61]:=(-1)*REAL_TO_WORD(65536-GVL.Chan1Ua*1000);	
			
	   END_IF
	   
	   IF GVL.Chan1Ue>0 THEN
			modbusInputRegs[62]:=REAL_TO_WORD(GVL.Chan1Ue*1000);
	   ELSE
			modbusInputRegs[62]:=(-1)*REAL_TO_WORD(65536-GVL.Chan1Ue*1000);	
			
	   END_IF
	   
			modbusInputRegs[63]:=REAL_TO_WORD(GVL.Chan2AGC*1000);
			modbusInputRegs[64]:=REAL_TO_WORD(GVL.Chan2Ua*1000);
			modbusInputRegs[65]:=REAL_TO_WORD(GVL.Chan2Ue*1000);
	ELSE
			modbusInputRegs[59]:=0;
			modbusInputRegs[60]:=0;
			modbusInputRegs[61]:=0;
			modbusInputRegs[62]:=0;
			modbusInputRegs[63]:=0;
			modbusInputRegs[64]:=0;
			modbusInputRegs[65]:=0;
	END_IF
	// =============================================================================
	// 段 E: 多项式程引系数 HR 解析（UnionLREAL_WORD，当前 RealTimePosCal 中已注释不用）
	// HR[71+] 各段 LREAL 系数，HR[335+] 节点时间；供 Get_AZ 备用路径
	// =============================================================================
	//IF GVL.AzCtrl.iMode = 11 AND GVL.ElCtrl.iMode = 11 THEN
	iCountPolyGet:=iCountPolyGet+1;
	//IF iCountPolyGet=10 THEN
		iCountPolyGet:=0;
	IF TRUE THEN
		FOR i := 0 TO 10 DO
			unionFun1_az[i].words[1] := modbusdata[74 + 4 * i];
			unionFun1_az[i].words[2] := modbusdata[73 + 4 * i];
			unionFun1_az[i].words[3] := modbusdata[72 + 4 * i];
			unionFun1_az[i].words[4] := modbusdata[71 + 4 * i];
			lrFun1_az[i] := unionFun1_az[i].lrealValue;
			
			unionFun2_az[i].words[1] := modbusdata[118 + 4 * i];
			unionFun2_az[i].words[2] := modbusdata[117 + 4 * i];
			unionFun2_az[i].words[3] := modbusdata[116 + 4 * i];
			unionFun2_az[i].words[4] := modbusdata[115 + 4 * i];
			lrFun2_az[i] := unionFun2_az[i].lrealValue;
			
			unionFun3_az[i].words[1] := modbusdata[162 + 4 * i];
			unionFun3_az[i].words[2] := modbusdata[161 + 4 * i];
			unionFun3_az[i].words[3] := modbusdata[160 + 4 * i];
			unionFun3_az[i].words[4] := modbusdata[159 + 4 * i];
			lrFun3_az[i] := unionFun3_az[i].lrealValue;
			
			unionFun4_az[i].words[1] := modbusdata[206 + 4 * i];
			unionFun4_az[i].words[2] := modbusdata[205 + 4 * i];
			unionFun4_az[i].words[3] := modbusdata[204 + 4 * i];
			unionFun4_az[i].words[4] := modbusdata[203 + 4 * i];
			lrFun4_az[i] := unionFun4_az[i].lrealValue;
			
			unionFun5_az[i].words[1] := modbusdata[250 + 4 * i];
			unionFun5_az[i].words[2] := modbusdata[249 + 4 * i];
			unionFun5_az[i].words[3] := modbusdata[248 + 4 * i];
			unionFun5_az[i].words[4] := modbusdata[247 + 4 * i];
			lrFun5_az[i] := unionFun5_az[i].lrealValue;
			
			unionFun6_az[i].words[1] := modbusdata[294 + 4 * i];
			unionFun6_az[i].words[2] := modbusdata[293 + 4 * i];
			unionFun6_az[i].words[3] := modbusdata[292 + 4 * i];
			unionFun6_az[i].words[4] := modbusdata[291 + 4 * i];
			lrFun6_az[i] := unionFun6_az[i].lrealValue;
			
			unionFun3_el[i].words[1] := modbusdata[450 + 4 * i];
			unionFun3_el[i].words[2] := modbusdata[449 + 4 * i];
			unionFun3_el[i].words[3] := modbusdata[448 + 4 * i];
			unionFun3_el[i].words[4] := modbusdata[447 + 4 * i];
			lrFun3_el[i] := unionFun3_el[i].lrealValue;
			
			unionFun4_el[i].words[1] := modbusdata[494 + 4 * i];
			unionFun4_el[i].words[2] := modbusdata[493 + 4 * i];
			unionFun4_el[i].words[3] := modbusdata[492 + 4 * i];
			unionFun4_el[i].words[4] := modbusdata[491 + 4 * i];
			lrFun4_el[i] := unionFun4_el[i].lrealValue;
			
			unionFun1_el[i].words[1] := modbusdata[362 + 4 * i];
			unionFun1_el[i].words[2] := modbusdata[361 + 4 * i];
			unionFun1_el[i].words[3] := modbusdata[360 + 4 * i];
			unionFun1_el[i].words[4] := modbusdata[359 + 4 * i];
			lrFun1_el[i] := unionFun1_el[i].lrealValue;
			
			unionFun2_el[i].words[1] := modbusdata[406 + 4 * i];
			unionFun2_el[i].words[2] := modbusdata[405 + 4 * i];
			unionFun2_el[i].words[3] := modbusdata[404 + 4 * i];
			unionFun2_el[i].words[4] := modbusdata[403 + 4 * i];
			lrFun2_el[i] := unionFun2_el[i].lrealValue;
			
			unionFun5_el[i].words[1] := modbusdata[538 + 4 * i];
			unionFun5_el[i].words[2] := modbusdata[537 + 4 * i];
			unionFun5_el[i].words[3] := modbusdata[536 + 4 * i];
			unionFun5_el[i].words[4] := modbusdata[535 + 4 * i];
			lrFun5_el[i] := unionFun5_el[i].lrealValue;
			
			unionFun6_el[i].words[1] := modbusdata[582 + 4 * i];
			unionFun6_el[i].words[2] := modbusdata[581 + 4 * i];
			unionFun6_el[i].words[3] := modbusdata[580 + 4 * i];
			unionFun6_el[i].words[4] := modbusdata[579 + 4 * i];
			lrFun6_el[i] := unionFun6_el[i].lrealValue;
		END_FOR
		i:=0;
		unionNodeTime1_az.words[1] := modbusdata[338];
		unionNodeTime1_az.words[2] := modbusdata[337];
		unionNodeTime1_az.words[3] := modbusdata[336];
		unionNodeTime1_az.words[4] := modbusdata[335];
		rNodeTime1_az := unionNodeTime1_az.lrealValue;
		
		unionNodeTime2_az.words[1] := modbusdata[342];
		unionNodeTime2_az.words[2] := modbusdata[341];
		unionNodeTime2_az.words[3] := modbusdata[340];
		unionNodeTime2_az.words[4] := modbusdata[339];
		rNodeTime2_az := unionNodeTime2_az.lrealValue;
		
		unionNodeTime3_az.words[1] := modbusdata[346];
		unionNodeTime3_az.words[2] := modbusdata[345];
		unionNodeTime3_az.words[3] := modbusdata[344];
		unionNodeTime3_az.words[4] := modbusdata[343];
		rNodeTime3_az := unionNodeTime3_az.lrealValue;
		
		unionNodeTime4_az.words[1] := modbusdata[350];
		unionNodeTime4_az.words[2] := modbusdata[349];
		unionNodeTime4_az.words[3] := modbusdata[348];
		unionNodeTime4_az.words[4] := modbusdata[347];
		rNodeTime4_az := unionNodeTime4_az.lrealValue;
		
		unionNodeTime5_az.words[1] := modbusdata[354];
		unionNodeTime5_az.words[2] := modbusdata[353];
		unionNodeTime5_az.words[3] := modbusdata[352];
		unionNodeTime5_az.words[4] := modbusdata[351];
		rNodeTime5_az := unionNodeTime5_az.lrealValue;

		unionStartTime.words[1]:=modbusdata[646];
		unionStartTime.words[2]:=modbusdata[645];
		unionStartTime.words[3]:=modbusdata[644];
		unionStartTime.words[4]:=modbusdata[643];
		starttime:=unionStartTime.lrealValue;
		unionEndTime.words[1] := modbusdata[358];
		unionEndTime.words[2] := modbusdata[357];
		unionEndTime.words[3] := modbusdata[356];
		unionEndTime.words[4] := modbusdata[355];
		rEndTime := unionEndTime.lrealValue;
		
		//FOR i := 0 TO 5 DO
			
		//END_FOR
		
		unionNodeTime1_el.words[1] := modbusdata[626];
		unionNodeTime1_el.words[2] := modbusdata[625];
		unionNodeTime1_el.words[3] := modbusdata[624];
		unionNodeTime1_el.words[4] := modbusdata[623];
		rNodeTime1_el := unionNodeTime1_el.lrealValue;
		
		unionNodeTime2_el.words[1] := modbusdata[630];
		unionNodeTime2_el.words[2] := modbusdata[629];
		unionNodeTime2_el.words[3] := modbusdata[628];
		unionNodeTime2_el.words[4] := modbusdata[627];
		rNodeTime2_el := unionNodeTime2_el.lrealValue;
		
		unionNodeTime3_el.words[1] := modbusdata[634];
		unionNodeTime3_el.words[2] := modbusdata[633];
		unionNodeTime3_el.words[3] := modbusdata[632];
		unionNodeTime3_el.words[4] := modbusdata[631];
		rNodeTime3_el := unionNodeTime3_el.lrealValue;
		
		unionNodeTime4_el.words[1] := modbusdata[638];
		unionNodeTime4_el.words[2] := modbusdata[637];
		unionNodeTime4_el.words[3] := modbusdata[636];
		unionNodeTime4_el.words[4] := modbusdata[635];
		rNodeTime4_el := unionNodeTime4_el.lrealValue;
		
		unionNodeTime5_el.words[1] := modbusdata[642];
		unionNodeTime5_el.words[2] := modbusdata[641];
		unionNodeTime5_el.words[3] := modbusdata[640];
		unionNodeTime5_el.words[4] := modbusdata[639];
		rNodeTime5_el := unionNodeTime5_el.lrealValue;
		
		(*
		//验证上位机下发数据
		unionSum.words[1]:=modbusdata[650];
		unionSum.words[2]:=modbusdata[649];
		unionSum.words[3]:=modbusdata[648];
		unionSum.words[4]:=modbusdata[647];
		lrSum:=unionSum.lrealValue;
		
		lrSumlocal:=lrFun1_az[10]+lrFun2_az[10]+lrFun3_az[10]+lrFun4_az[10]+lrFun5_az[10]+lrFun6_az[10]
					+lrFun1_el[10]+lrFun2_el[10]+lrFun3_el[10]+lrFun4_el[10]+lrFun5_el[10]+lrFun6_el[10];
		*)
		
		IF NOT bNotFirst THEN
			bCheck := TRUE; // 接收系数完成 开始检测 检测一次
		END_IF
		bNotFirst := TRUE;
	ELSE // 多项式相关变量清零
		bCheck := FALSE;
		bNotFirst := FALSE;
		rNodeTime1_az := 0.0;
		rNodeTime2_az := 0.0;
		rNodeTime3_az := 0.0;
		rNodeTime4_az := 0.0;
		rNodeTime5_az := 0.0;
		rEndTime := 0.0;
		
		FOR i := 0 TO 10 DO
			lrFun1_az[i] := 0;
			lrFun2_az[i] := 0;
			lrFun3_az[i] := 0;
			lrFun4_az[i] := 0;
			lrFun5_az[i] := 0;
			lrFun6_az[i] := 0;
			lrFun3_el[i] := 0;
			lrFun4_el[i] := 0;
		END_FOR
		
		rNodeTime1_el := 0;
		rNodeTime2_el := 0;
		rNodeTime3_el := 0;
		rNodeTime4_el := 0;
		rNodeTime5_el := 0;
		
		FOR i := 0 TO 5 DO
			lrFun1_el[i] := 0;
			lrFun2_el[i] := 0;
			lrFun5_el[i] := 0;
			lrFun6_el[i] := 0;
		END_FOR
	END_IF
	
END_IF

                  
END_PROGRAM

PROGRAM Az_ctrl_1
  VAR
    Axis2_Ctrl : Az_Ctrl_FB;  (* 方位轴控制 FB *)
    bRemote2LocalStop : BOOL;
    bLocal2RemoteStop : BOOL;
    Error : INT;
    Axis2Limit_pos : REAL;  (* 硬限位 +275° *)
    Axis2Limit_Neg : REAL;  (* 硬限位 -275° *)
    bRTriger : Standard.R_TRIG;
    bFTriger : Standard.F_TRIG;
    Stop2_Count : INT;
    bStop_2 : BOOL;  (* 方位轴停稳标志 *)
    rPosModeStepBias : LREAL;
    rPosModeStep : LREAL;
    rStepBiasMax : LREAL;
    rStepBias : LREAL;  (* Modbus rBias_2 逐步逼近 *)
    rStep : LREAL;
    rAuToStepBias : LREAL;
    rAuToStepBiasTemp : LREAL;
    rAutoStep : LREAL;
    TbAutoTrigger : Standard.F_TRIG;
    RbAutoTrigger : Standard.R_TRIG;
    rAutoTrackingBiasMax : LREAL;
    rLocalInitPosModeSpeed : REAL;
    rRemoteInitPosModeSpeed : REAL;
    iCountOffAuto : INT;
    iCasePBAutoTrack : INT;
    rKAuToStepBias : LREAL;
    bVisError : BOOL;  (* 全局 Error_code≠0 时 TRUE（可视化） *)
    a : INT;  (* 占位变量 a:=2（无功能影响） *)
    agcmaxsearch_tb : agcmaxsearch_pb_1;  (* 指向模式 AGC 搜索 *)
    rSearchNextStepTarget_tb : REAL;
    agcmaxsearch_pb : agcmaxsearch_pb_1;  (* 程引模式 AGC 搜索 *)
    rElthreshold : REAL;  (* 俯仰角门限：程引 AGC 搜索需 El-90° > 此值 *)
    toN1 : Standard.Ton;
    ttime1 : TIME;
    bstartagcmaxsearch : BOOL;
    rSearchNextStepTarget : REAL;
    rMaxPosTest : REAL;
    iCountSearch : UINT;
    iCountn : UINT;
    bstartSearchAz : BOOL;  (* 触发方位轴 AGC 螺旋搜索 *)
    bstartSearchEl : BOOL;  (* 触发俯仰轴 AGC 搜索（供 El_ctrl_1 使用） *)
    iCircly : INT;
    rAZSearchThr : REAL;
    rElSearchThr : REAL;
  END_VAR

                    (*==============================================================================
  PRG: Az_ctrl_1（方位轴 Az 顶层程序）
  任务: Canopen 10ms
  作用: 与 El_ctrl_1 对称，负责方位轴反馈、状态、自跟踪、AGC 搜索及 Az_Ctrl_FB 调用
  特点:
    - 软限位 ±275°；程引目标 rInterAzPos
    - 自跟踪用 AutoTrackingCal.rChanUa（方位误差，符号与俯仰相反）
    - 含螺旋/联合搜索触发: bstartSearchAz, bstartSearchEl（供俯仰 AGC 搜索联动）
    - rPIDCmdPos 中 SECURITYCHECK.AZ_out 为减号（与俯仰 el_out 加号不同）
==============================================================================*)


a := 2;  // 无业务含义，保持原逻辑
IF GVL.Error_code <> 0 THEN
	bVisError := TRUE;
ELSE
	bVisError := FALSE;
END_IF

(* 远控参量曾在此直赋，现由 Modbus_Slave 统一写入 Axis2Remote *)

// =============================================================================
// 段 1: 驱动状态 → Axis2Status
// =============================================================================
Axis2Status.Error := GVL.bAzStsBit3;
Axis2Status.ErrorID := GVL.eAzErrorcode;
Axis2Status.bServo_Enable := GVL.bAzStsBit0 AND GVL.bAzStsBit1 AND GVL.bAzStsBit2;
Axis2Status.bBrake := NOT (GVL.bAzStsBit0 AND GVL.bAzStsBit1 AND GVL.bAzStsBit2);
Axis2Status.Disabled := NOT (GVL.bAzStsBit0 AND GVL.bAzStsBit1 AND GVL.bAzStsBit2);
Axis2Remote.rSoft_limit_Negative:=-275;Axis2Remote.rSoft_limit_Postive:=275;
Axis2Local.rSoft_limit_Negative:=-275;Axis2Local.rSoft_limit_Postive:=275;

// =============================================================================
// 段 2: CANopen 反馈 → rFctVelReal_2 / rFctPosReal_2（方位无额外偏移）
// =============================================================================
rFctVelReal_2:=DINT_TO_REAL(diAzActVel)/524288.0*360.0;
rFctPosReal_2:=DINT_TO_REAL(diAzActPos)/524288.0*360.0;

// =============================================================================
// 段 3: rPosCmd 硬限位 ±275°
// =============================================================================
Axis2Limit_pos:=275;
Axis2Limit_Neg:=-275;
IF Axis2Remote.rPosCmd>Axis2Limit_pos THEN
	Axis2Remote.rPosCmd:=275;
ELSIF Axis2Remote.rPosCmd<Axis2Limit_Neg THEN
	 Axis2Remote.rPosCmd:=-275;  
END_IF

IF Axis2Local.rPosCmd>Axis2Limit_pos THEN
	Axis2Local.rPosCmd:=275;
ELSIF Axis2Local.rPosCmd<Axis2Limit_Neg THEN
	 Axis2Local.rPosCmd:=-275;  
END_IF

// =============================================================================
// 段 4: 停稳判定 → Axis2Status.Moving
// =============================================================================
IF  ABS(rFctVelReal_2)<0.035 THEN
	Stop2_Count:=Stop2_Count+1;
	IF Stop2_Count>100 THEN
		Stop2_Count:=101;
		bStop_2:=TRUE;;
	END_IF
ELSE
	Stop2_Count:=0;
	bStop_2:=FALSE;
END_IF
Axis2Status.Moving := NOT bStop_2;

// =============================================================================
// 段 5: PID 使能（mode 2 / 4）
// =============================================================================
IF Axis2Remote.iMode=2 OR Axis2Remote.iMode=4 THEN
	Axis2Remote.bPIDEnable:=TRUE;
ELSE
	Axis2Remote.bPIDEnable:=FALSE;
END_IF

// =============================================================================
// 段 6: 远控 ↔ 本控 切换保护（与 El 相同，halt=7 → 停稳 → powerOff=0）
// =============================================================================
bRTriger(CLK:=GVL.bLocalCtrl);
bFTriger(CLK:=GVL.bLocalCtrl);

IF Axis2Status.bServo_Enable AND (bRTriger.Q ) THEN//如果速度不为0且本控发生切换，则减速停止标识为True
	bRemote2LocalStop:=TRUE;
END_IF
IF bRemote2LocalStop  THEN //若减速停止标识符为True 
	
	IF  bStop_2=TRUE THEN//且电机速度不为0 开始减速 减速完成后下使能，下使能完成后复位标识符复位
		Axis2Local.iMode:=0;
		Axis2Remote.iMode:=0;
		IF Axis2Status.bServo_Enable=FALSE THEN
			bRemote2LocalStop:=FALSE;
		END_IF
	ELSE
		Axis2Local.iMode:=7;
		Axis2Remote.iMode:=7;
	END_IF
END_IF

IF Axis2Status.bServo_Enable AND (bFTriger.Q ) THEN//如果速度不为0且本控发生切换，则减速停止标识为True
	bLocal2RemoteStop:=TRUE;
END_IF
IF bLocal2RemoteStop  THEN //若减速停止标识符为True 
	
	IF  bStop_2=TRUE THEN//且电机速度不为0 开始减速 减速完成后下使能，下使能完成后复位标识符复位
		Axis2Local.iMode:=0;
		Axis2Remote.iMode:=0;
		IF Axis2Status.bServo_Enable=FALSE THEN
			bLocal2RemoteStop:=FALSE;
		END_IF
	ELSE
		Axis2Remote.iMode:=7;
		Axis2Local.iMode:=7;
	END_IF
END_IF

// =============================================================================
// 段 7: AGC 峰值搜索（bstart 来自 Modbus_slave.bSearch）
// mode2: rPosCmd；mode4: RealTimePosCal.rInterAzPos；需俯仰 El-90°>rElthreshold
// =============================================================================
IF Axis2Remote.iMode=2 THEN
			bstartagcmaxsearch:=Modbus_slave.bSearch;
			IF GVL.Chan1AGC>=(GVL.Chanthreshold-0.1) THEN
					agcmaxsearch_tb(bstart:=bstartagcmaxsearch,rAGCNow:=GVL.Chan1AGC,btrig:=bstartSearchAz,
				rinterPos:=Axis2Remote.rPosCmd,rcurrentpos:=GVL.rFctPosReal_2,
				rStepBiasNow:=0,bAutoTracking:=GVL.bStartTrack,bStop:=FALSE,
				rStepBias=>rSearchNextStepTarget_tb,rAGCMaxBias=>rMaxPosTest,bSucess=>);
			ELSE
				bstartagcmaxsearch:=FALSE;
				agcmaxsearch_tb(bstart:=bstartagcmaxsearch,rAGCNow:=GVL.Chan1AGC,btrig:=bstartSearchAz,
				rinterPos:=Axis2Remote.rPosCmd,rcurrentpos:=GVL.rFctPosReal_2,
				rStepBiasNow:=0,bAutoTracking:=GVL.bStartTrack,bStop:=FALSE,
				rStepBias=>rSearchNextStepTarget_tb,rAGCMaxBias=>rMaxPosTest,bSucess=>);
			END_IF
		ELSIF Axis2Remote.iMode=4 AND (GVL.rFctPosReal_1 - 90)>rElthreshold  THEN
			bstartagcmaxsearch:=Modbus_slave.bSearch;
			IF GVL.Chan1AGC>=(GVL.Chanthreshold-0.1) THEN
					agcmaxsearch_pb(bstart:=bstartagcmaxsearch,rAGCNow:=GVL.Chan1AGC,btrig:=bstartSearchAz,
				rinterPos:=RealTimeposcal.rInterAzPos,rcurrentpos:=GVL.rFctPosReal_2,
				rStepBiasNow:=rStepBias,bAutoTracking:=GVL.bStartTrack,bStop:=FALSE,
				rStepBias=>rSearchNextStepTarget,rAGCMaxBias=>rMaxPosTest,bSucess=>);
			ELSE
				bstartagcmaxsearch:=FALSE;
				agcmaxsearch_pb(bstart:=bstartagcmaxsearch,rAGCNow:=GVL.Chan1AGC,btrig:=bstartSearchAz,
				rinterPos:=RealTimeposcal.rInterAzPos,rcurrentpos:=GVL.rFctPosReal_2,
				rStepBiasNow:=rStepBias,bAutoTracking:=GVL.bStartTrack,bStop:=FALSE,
				rStepBias=>rSearchNextStepTarget,rAGCMaxBias=>rMaxPosTest,bSucess=>);
			END_IF
		ELSIF Axis2Remote.iMode =0  OR Axis2Remote.iMode =7 THEN
			bstartagcmaxsearch:=FALSE;
			iCountSearch:=0;
			agcmaxsearch_pb(bstart:=bstartagcmaxsearch,rAGCNow:=GVL.Chan1AGC,btrig:=bstartSearchAz,
			rinterPos:=RealTimeposcal.rInterAzPos,rcurrentpos:=GVL.rFctPosReal_2,
			rStepBiasNow:=rStepBias,bAutoTracking:=GVL.bStartTrack,bStop:=FALSE,
			rStepBias=>rSearchNextStepTarget,rAGCMaxBias=>rMaxPosTest,bSucess=>);
		END_IF
		
// =============================================================================
// 段 8: 自跟踪拉偏（远控）— 方位用 rChanUa，程引时符号与俯仰相反
// =============================================================================
IF GVL.bStartTrack AND Axis2Remote.iMode=4 THEN
	Axis2Remote.bStartAutoTrack := TRUE;
	IF rAuToStepBias > rAutoTrackingBiasMax THEN
		rAuToStepBias := rAutoTrackingBiasMax;
	ELSIF rAuToStepBias < -rAutoTrackingBiasMax THEN
		rAuToStepBias := -rAutoTrackingBiasMax;
	ELSE
		rAuToStepBiasTemp:=(-0.04)*AutoTrackingCal.rDirSenFac*AutoTrackingCal.rChanUa;
		rAuToStepBias:=rAuToStepBias-AutoTrackingCal.rDirSenFac*rKAuToStepBias*AutoTrackingCal.rChanUa/1000.0;
	END_IF
ELSIF NOT GVL.bStartTrack AND Axis2Remote.iMode=4 THEN
	IF 	rAuToStepBias>0 THEN//关闭自跟踪后自跟踪拉偏量逐渐归0
		rAuToStepBias:=rAuToStepBias-rAutoStep;
	ELSIF rAuToStepBias<0 THEN
		rAuToStepBias:=rAuToStepBias+rAutoStep;
	ELSE
		rAuToStepBias:=0;
	END_IF
	
	IF Modbus_Slave.rBias_2>rStepBias THEN
		rStepBias:=rStepBias+rStep;
		IF rStepBias>=Modbus_Slave.rBias_2 THEN
			rStepBias:=Modbus_Slave.rBias_2;
		END_IF
	ELSIF Modbus_Slave.rBias_2<rStepBias THEN
		rStepBias:=rStepBias-rStep;
		IF rStepBias<=Modbus_Slave.rBias_2 THEN
			rStepBias:=Modbus_Slave.rBias_2;
		END_IF
	END_IF
	rAuToStepBiasTemp:=0;
ELSIF GVL.bStartTrack AND Axis2Remote.iMode=2 THEN
	Axis2Remote.bStartAutoTrack := TRUE;
	Axis2Remote.rChanU := -AutoTrackingCal.rChanUa;
ELSE
	Axis2Remote.bStartAutoTrack := FALSE;	
	rAuToStepBias:=0;
	rStepBias:=0;
	rAuToStepBiasTemp:=0;
END_IF

// 本控自跟踪
IF GVL.bStartLocalAutoTrack AND Axis2Local.iMode = 4 THEN
	Axis2Local.bStartAutoTrack := TRUE;
	Axis2Local.rChanU := -AutoTrackingCal.rChanUaLocal;
ELSE
	Axis2Local.bStartAutoTrack := FALSE;
END_IF

// =============================================================================
// 段 9: 合成 rPIDCmdPos（注意 AZ_out 为减）→ Az_Ctrl_FB
// =============================================================================
Axis2Remote.rPIDCmdPos:=RealTimePosCal.rInterAzPos+rStepBias+rAuToStepBias+rSearchNextStepTarget-SECURITYCHECK.AZ_out+rAuToStepBiasTemp;

IF Axis2Remote.rPIDCmdPos<-275 THEN
	Axis2Remote.rPIDCmdPos:=-275;
ELSIF Axis2Remote.rPIDCmdPos>275 THEN
	Axis2Remote.rPIDCmdPos:=275;
END_IF

Axis2_Ctrl(sLocal:=Axis2Local, sCtrl:=Axis2Remote, sStatus:=Axis2Status, sVisible:=Axis2Visible, rRealPos:=rFctPosReal_2, rPosLimK:=0.34);

                  
END_PROGRAM

FUNCTION_BLOCK Az_Ctrl_FB
  VAR_INPUT
    sLocal : AxisCrtlStruct;  (* 本控命令结构体 *)
    sCtrl : AxisCrtlStruct;  (* 远控命令结构体 *)
    sStatus : AxisStatus;  (* 轴状态 *)
    sVisible : AxisVisible;  (* HMI 可视化（此 FB 未直接使用） *)
    rRealPos : REAL;  (* 编码器实际位置 (deg) *)
    rPosLimK : REAL;  (* 备用限位系数 *)
  END_VAR
  VAR_OUTPUT
    logicError : INT;  (* 保留 *)
  END_VAR
  VAR
    VelPID_1 : PID;  (* positionMode 用 *)
    VelPID_2 : PID;  (* 本控 programBootMode 用 *)
    VelPID_3 : PID;  (* 保留（已被 vpid1 替代） *)
    vpid1 : vpid;  (* 变增益 PID，programBootMode 远控 *)
    TON_0 : TON;  (* 超时 1s 强制下电计时器 *)
    bTick : BOOL;  (* stop0 超时标志 *)
    tr : BOOL;  (* 心跳恢复进行中标志 *)
    icount1 : INT;  (* 心跳恢复计数器1 *)
    icount2 : INT;  (* 心跳恢复计数器2 *)
    icount3 : INT;  (* 备用 *)
    bfin1 : BOOL;  (* 计数器1完成标志 *)
    bfin2 : BOOL;  (* 保留 *)
    istate : INT;  (* 上电状态机 *)
    icount : INT;  (* 上电步骤计数 *)
  END_VAR

                    (*==============================================================================
  FB: Az_Ctrl_FB（方位轴 Azimuth 控制功能块）
  与 El_Ctrl_FB 结构完全相同，差异点:
    - 操作的 GVL 变量为 Az 系列（diAzTargetVel / bAzCtrlBitX / eAzErrorcode 等）
    - positionMode 加速度为 12 deg/s²（El 为 9 deg/s²）
    - positionMode 的 Kp=0.6（El 为 0.7），本控 programBootMode Kp=0.6
    - programBootMode 参数来自 PersistentVars.rAzXxx

  速度换算公式（通用）:
    diAzTargetVel [inc/s] = deg/s × 524288 / 360
==============================================================================*)

// =============================================================================
// 段 A: 轴停止或下电时清快速停止位 bit8
// =============================================================================
IF sStatus.Disabled OR(NOT sStatus.Moving)THEN
	bAzCtrlBit8 := FALSE;
END_IF

// =============================================================================
// 段 B: 全局错误复位
// =============================================================================
IF GVL.bError_Reset THEN
	sCtrl.iMode:=6;
	sLocal.iMode:=6;
	GVL.Error_code:=0;
END_IF
IF GVL.Error_code =0 THEN
	GVL.bError_Reset:=FALSE;
END_IF

// =============================================================================
// 段 C: CANopen 心跳超时（0x8130）自动恢复序列
// =============================================================================
IF GVL.eAzErrorcode = 16#8130 AND NOT tr THEN
	GVL.bAzCtrlBit7 := TRUE;
	tr:=TRUE;
	istate:=0;
	icount:=0;
	// 写入下电控制字
	GVL.bAzCtrlBit3 := FALSE;
	GVL.bAzCtrlBit0 := FALSE;
	GVL.bAzCtrlBit1 := FALSE;
	GVL.bAzCtrlBit2 := FALSE;
END_IF
IF tr THEN
	icount1 := icount1 + 1;
END_IF
IF icount1 > 101 THEN
	icount1 := 0;
	tr := FALSE;
	GVL.bAzCtrlBit7 := FALSE;
	bfin1 := TRUE;
END_IF
IF bfin1 THEN
	icount2 := icount2 + 1;
END_IF
IF icount2 > 101 THEN
	bfin1 := FALSE;
	icount2 := 0;
END_IF

// =============================================================================
// 段 D: 主控制逻辑
// =============================================================================
IF GVL.Error_code=0 AND GVL.eAzErrorcode = 0 AND NOT GVL.bAzCtrlBit7  AND NOT tr AND NOT bfin1 AND NOT bfin2 THEN

	// =========== 远控 ===========
	IF GVL.bLocalCtrl=FALSE THEN //远控
		IF sCtrl.iMode <> 1 THEN
			istate:=0;
			icount:=0;
		END_IF
		CASE sCtrl.iMode OF

			MODES.powerOff: // 下电
				IF NOT sStatus.Disabled THEN
					IF sStatus.Moving THEN // 运动中，先停止运动
						GVL.diAzTargetVel := 0;
						bAzCtrlBit8 := TRUE;
					ELSE
						// 写入下电控制字
						GVL.bAzCtrlBit3 := FALSE;
						GVL.bAzCtrlBit0 := FALSE;
						GVL.bAzCtrlBit1 := FALSE;
						GVL.bAzCtrlBit2 := FALSE;
					END_IF
				END_IF
				// 下电状态下持续调用 vpid1（保持内部状态稳定）
				vpid1(rKpbase:=1, rKibase:=0.01, rKpMax:=1, rKiMax:=0.01, rVelThreshold:=10,rTarget:=sCtrl.rPIDCmdPos,rFeedback:=rRealPos,rPosLimPositive:=sCtrl.rSoft_limit_Postive,
							rPosLimNegitive:=sCtrl.rSoft_limit_Negative,
								bPIDEnable:=sCtrl.bPIDEnable,rVelLim:=sCtrl.rVel_Limit,rKpScale:=0.02,rKiScale:=0.005,rElPos:=GVL.rFctPosReal_1-90,
								iThrehold:=sCtrl.rPIDThre,rPIDOutDir=>sCtrl.rPIDCmdVel);

			MODES.powerOn:  // 上电（DS402 三步序列）
				IF sStatus.Disabled THEN
					GVL.diAzTargetVel := 0;
					IF GVL.siAzMode <> 3 THEN // 上电时模式默认为3，速度模式
						GVL.siAzMode := 3;
					END_IF
					IF siAzMode = 3 THEN
						CASE istate OF
							0:
								GVL.bAzCtrlBit1 := TRUE;
								GVL.bAzCtrlBit2 := TRUE;
								icount := icount + 1;
								IF icount = 20 THEN
									icount:=0;
									istate:=1;
								END_IF
							1:
								GVL.bAzCtrlBit0 := TRUE;
								icount := icount + 1;
								IF icount = 20 THEN
									icount:=0;
									istate:=2;
								END_IF
							2:
								GVL.bAzCtrlBit3 := TRUE;
						END_CASE
					END_IF
				ELSE
					IF sStatus.Moving THEN
						GVL.diAzTargetVel := 0;
						bAzCtrlBit8 := TRUE;
					ELSE
						bAzCtrlBit8 := FALSE;
					END_IF
				END_IF

			MODES.positionMode: // 远控指向模式（加速度 12 deg/s²，Kp=0.6）
				IF NOT sStatus.Disabled THEN
					IF sCtrl.bStartAutoTrack THEN
						//自跟踪模式下，由误差电压直接驱动
						VelPID_1(rTarget:=sCtrl.rChanU + rRealPos,
								rFeedback:=rRealPos,
								rPosLimPositive:=sCtrl.rSoft_limit_Postive,
								rPosLimNegative:=sCtrl.rSoft_limit_Negative,
								rVelLim:=sCtrl.rVel_Limit,
								rKp:=1,//自跟踪PI系数3,0.02
								rKi:=0,
								rKd:=0,
								bPIDEnable:=sCtrl.bPIDEnable,
								iThreshold:= -1,
								rPIDOutput=>sCtrl.rPIDCmdVel);							
					ELSE
						//PID计算速度指令
						VelPID_1(rTarget:=sCtrl.rPosCmd,
							rFeedback:=rRealPos,
							rVelLim:=sCtrl.Pos_Vel,
							rPosLimPositive:=sCtrl.rSoft_limit_Postive,
							rPosLimNegative:=sCtrl.rSoft_limit_Negative,
							rKp:=0.6,//程引PI系数低带：1,0.002  高带：3,0.02
							rKi:=0,
							rKd:=0,
							bPIDEnable:=sCtrl.bPIDEnable,
							iThreshold:=sCtrl.rPIDThre,
							rPIDOutput=>sCtrl.rPIDCmdVel);
					END_IF
					GVL.diAzTargetVel := REAL_TO_DINT(sCtrl.rPIDCmdVel * 524288 / 360);
					GVL.diAzTargetAcc := REAL_TO_UDINT(12 * 524288 / 360);   //加速度 12 deg/s²
					GVL.diAzTargetDec := REAL_TO_UDINT(12 * 524288 / 360);   //减速度
				END_IF

			MODES.velocityMode://手控速度模式-远控模式
				IF NOT sStatus.Disabled THEN
					IF ABS(sCtrl.rVelCmd) <= sCtrl.rVel_Limit THEN
						GVL.diAzTargetVel := REAL_TO_DINT(sCtrl.rVelCmd * 524288 / 360);
					ELSIF sCtrl.rVelCmd > sCtrl.rVel_Limit THEN
						GVL.diAzTargetVel := REAL_TO_DINT(sCtrl.rVel_Limit * 524288 / 360);
					ELSE
						GVL.diAzTargetVel := REAL_TO_DINT(-sCtrl.rVel_Limit * 524288 / 360);
					END_IF
					GVL.diAzTargetAcc := REAL_TO_UDINT(sCtrl.rAcceleration * 524288 / 360);   //加速度
					GVL.diAzTargetDec := REAL_TO_UDINT(sCtrl.rDeceleration * 524288 / 360);   //减速度
				END_IF

			MODES.programBootMode://PID速度模式-正常模式 程引（变增益 vpid1）
				IF NOT sStatus.Disabled THEN
					IF sCtrl.bStartAutoTrack THEN
						// 程引+自跟踪
						vpid1(rKpbase:=Persistentvars.rAzKpBase, rKibase:=Persistentvars.rAzKiBase, rKpMax:=Persistentvars.rAzKpMax, rKiMax:=Persistentvars.rAzKiMax, rVelThreshold:=Persistentvars.rAzThre,rTarget:=sCtrl.rPIDCmdPos,rFeedback:=rRealPos,rPosLimPositive:=sCtrl.rSoft_limit_Postive,
							rPosLimNegitive:=sCtrl.rSoft_limit_Negative,
								bPIDEnable:=sCtrl.bPIDEnable,rVelLim:=sCtrl.rVel_Limit,rKpScale:=Persistentvars.rAzKpscale,rKiScale:=Persistentvars.rAzKiscale,rElPos:=GVL.rFctPosReal_1-90,
								iThrehold:=sCtrl.rPIDThre,rPIDOutDir=>sCtrl.rPIDCmdVel);							
					ELSE
						// 纯程引
						vpid1(rKpbase:=Persistentvars.rAzKpBase, rKibase:=Persistentvars.rAzKiBase, rKpMax:=Persistentvars.rAzKpMax, rKiMax:=Persistentvars.rAzKiMax, rVelThreshold:=Persistentvars.rAzThre,rTarget:=sCtrl.rPIDCmdPos,rFeedback:=rRealPos,rPosLimPositive:=sCtrl.rSoft_limit_Postive,
							rPosLimNegitive:=sCtrl.rSoft_limit_Negative,
								bPIDEnable:=sCtrl.bPIDEnable,rVelLim:=sCtrl.rVel_Limit,rKpScale:=Persistentvars.rAzKpscale,rKiScale:=Persistentvars.rAzKiscale,rElPos:=GVL.rFctPosReal_1-90,
								iThrehold:=sCtrl.rPIDThre,rPIDOutDir=>sCtrl.rPIDCmdVel);
						
					END_IF
					GVL.diAzTargetVel := REAL_TO_DINT(sCtrl.rPIDCmdVel * 524288 / 360);
					GVL.diAzTargetAcc := REAL_TO_UDINT(sCtrl.rAcceleration * 524288 / 360);   //加速度
					GVL.diAzTargetDec := REAL_TO_UDINT(sCtrl.rDeceleration * 524288 / 360);   //减速度
				END_IF

			MODES.reset://重置
				IF NOT sStatus.Disabled THEN
					IF sStatus.Moving THEN
						GVL.diAzTargetVel := 0;
						bAzCtrlBit8 := TRUE;
					ELSE
						bAzCtrlBit8 := FALSE;
					END_IF
				END_IF

			MODES.halt://待机
				IF NOT sStatus.Disabled THEN
					IF sStatus.Moving THEN
						GVL.diAzTargetVel := 0;
						bAzCtrlBit8 := TRUE;
					ELSE
						bAzCtrlBit8 := FALSE;
					END_IF
				END_IF
			
		END_CASE

	// =========== 本控 ===========
	ELSE // 本控
		IF sLocal.iMode <> 1 THEN
			istate:=0;
			icount:=0;
		END_IF
		CASE sLocal.iMode OF

			MODES.powerOff: // 下电
				IF NOT sStatus.Disabled THEN
					IF sStatus.Moving THEN // 运动中，先停止运动
						GVL.diAzTargetVel := 0;
						bAzCtrlBit8 := TRUE;
					ELSE
						// 写入下电控制字
						GVL.bAzCtrlBit3 := FALSE;
						GVL.bAzCtrlBit0 := FALSE;
						GVL.bAzCtrlBit1 := FALSE;
						GVL.bAzCtrlBit2 := FALSE;
					END_IF
				END_IF

			MODES.powerOn:  // 上电
				IF sStatus.Disabled THEN
					GVL.diAzTargetVel := 0;
					IF GVL.siAzMode <> 3 THEN // 上电时模式默认为3，速度模式
						GVL.siAzMode := 3;
					END_IF
					IF siAzMode = 3 THEN
						CASE istate OF
							0:
								GVL.bAzCtrlBit1 := TRUE;
								GVL.bAzCtrlBit2 := TRUE;
								icount := icount + 1;
								IF icount = 20 THEN
									icount:=0;
									istate:=1;
								END_IF
							1:
								GVL.bAzCtrlBit0 := TRUE;
								icount := icount + 1;
								IF icount = 20 THEN
									icount:=0;
									istate:=2;
								END_IF
							2:
								GVL.bAzCtrlBit3 := TRUE;
						END_CASE
					END_IF
				ELSE
					IF sStatus.Moving THEN
						GVL.diAzTargetVel := 0;
						bAzCtrlBit8 := TRUE;
					ELSE
						bAzCtrlBit8 := FALSE;
					END_IF
				END_IF

			MODES.velocityMode://手控速度模式-本控模式
				IF NOT sStatus.Disabled THEN
					IF ABS(sLocal.rVelCmd) <= sLocal.rVel_Limit THEN
						GVL.diAzTargetVel := REAL_TO_DINT(sLocal.rVelCmd * 524288 / 360);
					ELSIF sLocal.rVelCmd > sLocal.rVel_Limit THEN
						GVL.diAzTargetVel := REAL_TO_DINT(sLocal.rVel_Limit * 524288 / 360);
					ELSE
						GVL.diAzTargetVel := REAL_TO_DINT(-sLocal.rVel_Limit * 524288 / 360);
					END_IF
					GVL.diAzTargetAcc := REAL_TO_UDINT(sLocal.rAcceleration * 524288 / 360);   //加速度
					GVL.diAzTargetDec := REAL_TO_UDINT(sLocal.rDeceleration * 524288 / 360);   //减速度
				END_IF

			MODES.programBootMode://本控位置模式（普通 PID，Kp=0.6）
				IF NOT sStatus.Disabled THEN
					IF NOT sLocal.bPIDEnable THEN
						GVL.diAzTargetVel := 0;							
					ELSE
						IF NOT slocal.bStartAutoTrack THEN
							//PID计算速度指令
							 VelPID_2(rTarget:=sLocal.rPosCmd,
									 rFeedback:=rRealPos,
									 rPosLimPositive:=sLocal.rSoft_limit_Postive,//软限位
									 rPosLimNegative:=sLocal.rSoft_limit_Negative,
									 rKp:=0.6,
									 rKi:=0,
									 rKd:=0,
									 iThreshold:=sLocal.rPIDThre,
									 bPIDEnable:=sLocal.bPIDEnable,
									 rVelLim:=sLocal.Pos_Vel,
									 rPIDOutput=>sLocal.rPIDCmdVel);//普通PID
						ELSE
							//PID计算速度指令
							 VelPID_2(rTarget:=sLocal.rChanU + rRealPos,
								rFeedback:=rRealPos,
								rPosLimPositive:=sLocal.rSoft_limit_Postive,
								rPosLimNegative:=sLocal.rSoft_limit_Negative,
								rVelLim:=sLocal.rVel_Limit,
								rKp:=1,//自跟踪PI系数3,0.02
								rKi:=0,
								rKd:=0,
								bPIDEnable:=sLocal.bPIDEnable,
								iThreshold:= -1,
								rPIDOutput=>sLocal.rPIDCmdVel);//普通PID
						END_IF
						
					END_IF
					GVL.diAzTargetVel := REAL_TO_DINT(sLocal.rPIDCmdVel * 524288 / 360);
					GVL.diAzTargetAcc := REAL_TO_UDINT(12 * 524288 / 360);   //加速度
					GVL.diAzTargetDec := REAL_TO_UDINT(12 * 524288 / 360);   //减速度
				END_IF

			MODES.reset://重置
			// 是否需要
			MODES.halt://待机
				IF NOT sStatus.Disabled THEN
					IF sStatus.Moving THEN
						GVL.diAzTargetVel := 0;
						bAzCtrlBit8 := TRUE;
					ELSE
						bAzCtrlBit8 := FALSE;
					END_IF
				END_IF
			
		END_CASE
	END_IF

// =============================================================================
// 段 E: 全局错误时强制停轴，超时后强制下电
// =============================================================================
ELSIF GVL.Error_code<>0 AND GVL.eAzErrorcode = 0 AND NOT GVL.bAzCtrlBit7  AND NOT tr AND NOT bfin1 AND NOT bfin2 THEN
	// 出现错误，轴停止运动
	GVL.diAzTargetVel := 0;
	bAzCtrlBit8 := TRUE;
	TON_0(IN:=bAzCtrlBit8,PT:=T#1S,Q=>,ET=>);//判断stop0执行是否超时,若超时强制下电（手动复位）
	IF TON_0.Q THEN
		bTick:=TRUE;
	END_IF
	IF bTick AND sStatus.Moving THEN // 超时强制下电
		// 写入下电控制字
		GVL.bAzCtrlBit3 := FALSE;
		GVL.bAzCtrlBit0 := FALSE;
		GVL.bAzCtrlBit1 := FALSE;
		GVL.bAzCtrlBit2 := FALSE;
	END_IF
END_IF

                  
END_FUNCTION_BLOCK

FUNCTION_BLOCK solvex
  VAR_IN_OUT
    M : ARRAY[1..3, 1..3] OF LREAL;  (* 定义3x3矩阵M *)
    G : ARRAY[1..3] OF LREAL;  (* 定义3x1数组G *)
  END_VAR
  VAR
    AdjointMatrix : ARRAY[1..3, 1..3] OF REAL;  (* 用于存储伴随矩阵 *)
    Determinant : REAL;  (* 行列式 *)
    i : INT;  (* M_Inverse: ARRAY [1..3, 1..3] OF REAL; //逆矩阵 *)
    j : INT;  (* M_Inverse: ARRAY [1..3, 1..3] OF REAL; //逆矩阵 *)
    k : INT;  (* M_Inverse: ARRAY [1..3, 1..3] OF REAL; //逆矩阵 *)
    Temp : REAL;
  END_VAR
  VAR_OUTPUT
    X : ARRAY[1..3] OF REAL;  (* 用于存储解x *)
  END_VAR

                    
// 计算矩阵的行列式
Determinant := M[1, 1] * (M[2, 2] * M[3, 3] - M[2, 3] * M[3, 2]) -
               M[1, 2] * (M[2, 1] * M[3, 3] - M[2, 3] * M[3, 1]) +
               M[1, 3] * (M[2, 1] * M[3, 2] - M[2, 2] * M[3, 1]);

(*
// 计算3x3矩阵的伴随矩阵
Determinant := M[1, 1] * (M[2, 2] * M[3, 3] - M[2, 3] * M[3, 2]) -
               M[1, 2] * (M[2, 1] * M[3, 3] - M[2, 3] * M[3, 1]) +
               M[1, 3] * (M[2, 1] * M[3, 2] - M[2, 2] * M[3, 1]);

IF ABS(Determinant) > 1.0E-6 THEN
    FOR i := 1 TO 3 DO
        FOR j := 1 TO 3 DO
            AdjointMatrix[i, j] := M[(i MOD 3) + 1, (j MOD 3) + 1] * M[((i + 1) MOD 3) + 1, ((j + 1) MOD 3) + 1] -
                                   M[(i MOD 3) + 1, ((j + 1) MOD 3) + 1] * M[((i + 1) MOD 3) + 1, (j MOD 3) + 1];
        END_FOR
    END_FOR

    FOR i := 1 TO 3 DO
        FOR j := 1 TO 3 DO
            AdjointMatrix[j, i] := AdjointMatrix[i, j];
            AdjointMatrix[i, j] := AdjointMatrix[i, j] / Determinant;
        END_FOR
    END_FOR
END_IF
*)
// 计算3x3矩阵的伴随矩阵
Determinant := M[1, 1] * (M[2, 2] * M[3, 3] - M[2, 3] * M[3, 2]) -
               M[1, 2] * (M[2, 1] * M[3, 3] - M[2, 3] * M[3, 1]) +
               M[1, 3] * (M[2, 1] * M[3, 2] - M[2, 2] * M[3, 1]);

IF ABS(Determinant) > 1.0E-6 THEN
    FOR i := 1 TO 3 DO
        FOR j := 1 TO 3 DO
            AdjointMatrix[j, i] := ((M[(i MOD 3) + 1, (j MOD 3) + 1] * M[((i + 1) MOD 3) + 1, ((j + 1) MOD 3) + 1] -
                                   M[(i MOD 3) + 1, ((j + 1) MOD 3) + 1] * M[((i + 1) MOD 3) + 1, (j MOD 3) + 1]) / Determinant);
        END_FOR
    END_FOR
END_IF

// 计算X = AdjointMatrix * G
FOR i := 1 TO 3 DO
    X[i] := 0.0;
    FOR j := 1 TO 3 DO
        X[i] := X[i] + AdjointMatrix[i, j] * G[j];
    END_FOR
END_FOR




                  
END_FUNCTION_BLOCK

FUNCTION_BLOCK El_Ctrl_FB
  VAR_INPUT
    sLocal : AxisCrtlStruct;  (* 本控命令结构体（来自本地操作面板/GVL.sXxLocal） *)
    sCtrl : AxisCrtlStruct;  (* 远控命令结构体（来自 Modbus/上位机/GVL.sXxCtrl） *)
    sStatus : AxisStatus;  (* 轴状态（Disabled/Moving/Error 等标志） *)
    sVisible : AxisVisible;  (* HMI 可视化相关（此 FB 内部未直接使用） *)
    rRealPos : REAL;  (* 编码器实际位置 (deg)，即 GVL.rFctPosReal_X *)
    rPosLimK : REAL;  (* 备用限位系数（当前逻辑未使用） *)
  END_VAR
  VAR_OUTPUT
    logicError : INT;  (* 逻辑错误码（保留，当前未赋值） *)
  END_VAR
  VAR
    VelPID_1 : PID;  (* 位置模式（positionMode）用普通 PID *)
    VelPID_2 : PID;  (* 本控位置模式（programBootMode 本控）用普通 PID *)
    VelPID_3 : PID;  (* 保留（已被 vpid1 替代，代码中注释掉） *)
    vpid1 : vpid;  (* 变增益 PID，用于 programBootMode 远控/自跟踪 *)
    TON_0 : TON;  (* 延时 1s，错误时判断 stop0 是否超时 *)
    bTick : BOOL;  (* stop0 超时后置位，触发强制下电 *)
    tr : BOOL;  (* 心跳错误正在处理中标志（防止重入） *)
    icount1 : INT;  (* 心跳恢复计数器（等 101 拍 ≈ 1s 后清 bit7） *)
    icount2 : INT;  (* 清 bit7 后再等 101 拍才结束保护 *)
    icount3 : INT;  (* 备用 *)
    bfin1 : BOOL;  (* icount1 到达后置位，触发 icount2 阶段 *)
    bfin2 : BOOL;  (* 保留 *)
    istate : INT;  (* 上电序列状态机（0→1→2） *)
    icount : INT;  (* 上电序列各步骤等待计数（20 拍 = 200ms） *)
  END_VAR

                    
(*==============================================================================
  FB: El_Ctrl_FB（俯仰轴 Elevation 控制功能块）
  任务: Canopen 10ms（周期调用）
  作用:
    - 根据 sCtrl/sLocal 的 iMode，产生对应 CANopen 速度/控制字写入
    - 封装上/下电序列、软限位保护、CANopen 错误码自动恢复、心跳丢失处理
    - 内部调用 PID / vpid 进行位置→速度的闭环换算
  输入: sCtrl（远控命令结构体）、sLocal（本控命令结构体）
        sStatus（轴状态）、rRealPos（编码器实际角度）
  输出: 直接写 GVL.diElTargetVel / diElTargetAcc / diElTargetDec 及控制字位

  速度换算公式（通用）:
    diXxTargetVel [inc/s] = deg/s × 524288 / 360
    其中 524288 = 2^19（CANopen 电机编码器增量/转，具体由电机参数决定）
==============================================================================*)


// =============================================================================
// 段 A: 全局复位 — 轴停止或下电时清 bit8（快速停止位）
// bit8=1 激活快速停止，bit8=0 正常运行
// =============================================================================
IF sStatus.Disabled OR (NOT sStatus.Moving) THEN
	bElCtrlBit8 := FALSE;
END_IF

// =============================================================================
// 段 B: 错误复位（由 HMI 或 Modbus 写 bError_Reset）
// 将两个命令结构体模式设为 reset(6)，清 Error_code
// =============================================================================
IF GVL.bError_Reset THEN
	sCtrl.iMode:=6;
	sLocal.iMode:=6;
	GVL.Error_code:=0;
END_IF
IF GVL.Error_code =0 THEN
	GVL.bError_Reset:=FALSE;
END_IF

// =============================================================================
// 段 C: CANopen 心跳超时错误（错误码 0x8130）自动恢复序列
// 步骤: 设 bit7(故障复位位) → 等 101 拍 → 清 bit7 → 再等 101 拍 → 结束
// 期间同时下电（清控制字 bit0~3），待驱动自愈后再由上层重新上电
// =============================================================================
IF GVL.eElErrorcode = 16#8130 AND NOT tr THEN
	GVL.bElCtrlBit7 := TRUE;  // 触发驱动故障复位
	tr:=TRUE;
	istate:=0;
	icount:=0;
	// 写入下电控制字
	GVL.bElCtrlBit3 := FALSE;
	GVL.bElCtrlBit0 := FALSE;
	GVL.bElCtrlBit1 := FALSE;
	GVL.bElCtrlBit2 := FALSE;	
END_IF
IF tr THEN
	icount1 := icount1 + 1;
END_IF
IF icount1 > 101 THEN     // 约 1s（10ms × 101）后清故障复位位
	icount1 := 0;
	tr := FALSE;
	GVL.bElCtrlBit7 := FALSE;
	bfin1 := TRUE;
END_IF
IF bfin1 THEN             // 再等 1s 让驱动彻底稳定
	icount2 := icount2 + 1;
END_IF
IF icount2 > 101 THEN
	bfin1 := FALSE;
	icount2 := 0;
END_IF

// =============================================================================
// 段 D: 主控制逻辑
// 条件: 无全局错误 AND 无驱动错误 AND 不在心跳恢复序列中
// =============================================================================
IF GVL.Error_code=0 AND GVL.eElErrorcode = 0 AND NOT GVL.bElCtrlBit7  AND NOT tr AND NOT bfin1 AND NOT bfin2 THEN

	// =========== 远控分支（bLocalCtrl=FALSE） ===========
	IF GVL.bLocalCtrl=FALSE THEN //远控
		IF sCtrl.iMode <> 1 THEN   // 非上电模式时重置上电状态机
			istate:=0;
			icount:=0;
		END_IF
		CASE sCtrl.iMode OF

			// ----- 模式 0: 下电 -----
			MODES.powerOff: // 下电
				IF NOT sStatus.Disabled THEN
					IF sStatus.Moving THEN // 运动中，先停止运动
						GVL.diElTargetVel := 0;
						bElCtrlBit8 := TRUE;   // 发快速停止
					ELSE
						// 写入下电控制字（bit0~3=0 即断使能）
						GVL.bElCtrlBit3 := FALSE;
						GVL.bElCtrlBit0 := FALSE;
						GVL.bElCtrlBit1 := FALSE;
						GVL.bElCtrlBit2 := FALSE;
					END_IF
				END_IF
				// 注: 下电模式仍持续运行 vpid1，但输出不写到 diElTargetVel
				// 目的是让 vpid1 内部积分不要突变（实际速度已通过控制字停掉）
				vpid1(rKpbase:=1, rKibase:=0.01, rKpMax:=1, rKiMax:=0.01, rVelThreshold:=10,rTarget:=sCtrl.rPIDCmdPos,rFeedback:=rRealPos,rPosLimPositive:=sCtrl.rSoft_limit_Postive,
							rPosLimNegitive:=sCtrl.rSoft_limit_Negative,
								bPIDEnable:=sCtrl.bPIDEnable,rVelLim:=sCtrl.rVel_Limit,rKpScale:=0.02,rKiScale:=0.005,rElPos:=GVL.rFctPosReal_1-90,
								iThrehold:=sCtrl.rPIDThre,rPIDOutDir=>sCtrl.rPIDCmdVel);

			// ----- 模式 1: 上电（三步 CANopen DS402 状态机）-----
			MODES.powerOn:  // 上电
				IF sStatus.Disabled THEN
					GVL.diElTargetVel := 0;
					IF GVL.siElMode <> 3 THEN // 上电时模式默认为3，速度模式
						GVL.siElMode := 3;
					END_IF
					IF siElMode = 3 THEN
						// DS402 上电序列: Shutdown → Switch On → Enable Operation
						// 每步等待 20 拍（200ms）确保驱动应答
						CASE istate OF
							0:  // Shutdown: bit1=1, bit2=1（清故障 + 切换允许）
								GVL.bElCtrlBit1 := TRUE;
								GVL.bElCtrlBit2 := TRUE;
								icount := icount + 1;
								IF icount = 20 THEN
									icount:=0;
									istate:=1;
								END_IF
							1:  // Switch On: bit0=1
								GVL.bElCtrlBit0 := TRUE;
								icount := icount + 1;
								IF icount = 20 THEN
									icount:=0;
									istate:=2;
								END_IF
							2:  // Enable Operation: bit3=1
								GVL.bElCtrlBit3 := TRUE;
						END_CASE
					END_IF
				ELSE
					// 已上电：若还在运动则发快速停止等待停稳
					IF sStatus.Moving THEN
						GVL.diElTargetVel := 0;
						bElCtrlBit8 := TRUE;
					ELSE
						bElCtrlBit8 := FALSE;
					END_IF
				END_IF

			// ----- 模式 2: 指向模式（位置 PID 输出速度，远控）-----
			MODES.positionMode: // 远控指向模式
				IF NOT sStatus.Disabled THEN
					IF sCtrl.bStartAutoTrack THEN
						// 自跟踪模式：误差电压（rChanU）直接作为位置增量指令
						// 即: 目标 = rChanU（deg，来自跟踪接收机） + 当前位置
						VelPID_1(rTarget:=sCtrl.rChanU + rRealPos,
								rFeedback:=rRealPos,
								rPosLimPositive:=sCtrl.rSoft_limit_Postive,
								rPosLimNegative:=sCtrl.rSoft_limit_Negative,
								rVelLim:=sCtrl.rVel_Limit,
								rKp:=1,//自跟踪PI系数3,0.02
								rKi:=0,
								rKd:=0,
								bPIDEnable:=sCtrl.bPIDEnable,
								iThreshold:= -1,   // -1=始终开积分
								rPIDOutput=>sCtrl.rPIDCmdVel);							
					ELSE
						// 指向模式：目标为上位机给定的角度
						VelPID_1(rTarget:=sCtrl.rPosCmd,
							rFeedback:=rRealPos,
							rVelLim:=sCtrl.Pos_Vel,
							rPosLimPositive:=sCtrl.rSoft_limit_Postive,
							rPosLimNegative:=sCtrl.rSoft_limit_Negative,
							rKp:=0.7,//程引PI系数地带：1,0.002  高带：3,0.02
							rKi:=0,
							rKd:=0,
							bPIDEnable:=sCtrl.bPIDEnable,
							iThreshold:=sCtrl.rPIDThre,
							rPIDOutput=>sCtrl.rPIDCmdVel);
					END_IF
					// 将 PID 输出速度(deg/s)换算为 CANopen 速度增量单位写入
					GVL.diElTargetVel := REAL_TO_DINT(sCtrl.rPIDCmdVel * 524288 / 360);
					GVL.diElTargetAcc := REAL_TO_UDINT(9 * 524288 / 360);   //加速度 9 deg/s²
					GVL.diElTargetDec := REAL_TO_UDINT(9 * 524288 / 360);   //减速度
				END_IF

			// ----- 模式 3: 速度模式（手动点动，远控）-----
			MODES.velocityMode://手控速度模式-远控模式
				IF NOT sStatus.Disabled THEN
					// 限幅处理：超过限速则取限速值
					IF ABS(sCtrl.rVelCmd) <= sCtrl.rVel_Limit THEN
						GVL.diElTargetVel := REAL_TO_DINT(sCtrl.rVelCmd * 524288 / 360);
					ELSIF sCtrl.rVelCmd > sCtrl.rVel_Limit THEN
						GVL.diElTargetVel := REAL_TO_DINT(sCtrl.rVel_Limit * 524288 / 360);
					ELSE
						GVL.diElTargetVel := REAL_TO_DINT(-sCtrl.rVel_Limit * 524288 / 360);
					END_IF
					GVL.diElTargetAcc := REAL_TO_UDINT(sCtrl.rAcceleration * 524288 / 360);   //加速度
					GVL.diElTargetDec := REAL_TO_UDINT(sCtrl.rDeceleration * 524288 / 360);   //减速度
				END_IF

			// ----- 模式 4: 程引模式（程序引导/插值跟踪，远控）-----
			// 使用变增益 vpid1，参数来自 PersistentVars（标定可调）
			MODES.programBootMode://PID速度模式-正常模式 程引
				IF NOT sStatus.Disabled THEN
					IF sCtrl.bStartAutoTrack THEN
						// 程引+自跟踪：误差电压叠加到插值目标位置上
						vpid1(rKpbase:=Persistentvars.rElKpBase, rKibase:=Persistentvars.rElKiBase, rKpMax:=Persistentvars.rElKpMax, rKiMax:=Persistentvars.rElKiMax, rVelThreshold:=Persistentvars.rElThre,rTarget:=sCtrl.rPIDCmdPos,rFeedback:=rRealPos,rPosLimPositive:=sCtrl.rSoft_limit_Postive,
							rPosLimNegitive:=sCtrl.rSoft_limit_Negative,
								bPIDEnable:=sCtrl.bPIDEnable,rVelLim:=sCtrl.rVel_Limit,rKpScale:=Persistentvars.rElKpscale,rKiScale:=Persistentvars.rElKiscale,rElPos:=GVL.rFctPosReal_1-90,
								iThrehold:=sCtrl.rPIDThre,rPIDOutDir=>sCtrl.rPIDCmdVel);						
					ELSE
						// 程引不开自跟踪：纯插值位置跟踪
						vpid1(rKpbase:=Persistentvars.rElKpBase, rKibase:=Persistentvars.rElKiBase, rKpMax:=Persistentvars.rElKpMax, rKiMax:=Persistentvars.rElKiMax, rVelThreshold:=Persistentvars.rElThre,rTarget:=sCtrl.rPIDCmdPos,rFeedback:=rRealPos,rPosLimPositive:=sCtrl.rSoft_limit_Postive,
							rPosLimNegitive:=sCtrl.rSoft_limit_Negative,
								bPIDEnable:=sCtrl.bPIDEnable,rVelLim:=sCtrl.rVel_Limit,rKpScale:=Persistentvars.rElKpscale,rKiScale:=Persistentvars.rElKiscale,rElPos:=GVL.rFctPosReal_1-90,
								iThrehold:=sCtrl.rPIDThre,rPIDOutDir=>sCtrl.rPIDCmdVel);
					END_IF
					GVL.diElTargetVel := REAL_TO_DINT(sCtrl.rPIDCmdVel * 524288 / 360);
					GVL.diElTargetAcc := REAL_TO_UDINT(sCtrl.rAcceleration * 524288 / 360);   //加速度
					GVL.diElTargetDec := REAL_TO_UDINT(sCtrl.rDeceleration * 524288 / 360);   //减速度
				END_IF

			// ----- 模式 6: 重置 -----
			MODES.reset://重置
				IF NOT sStatus.Disabled THEN
					IF sStatus.Moving THEN
						GVL.diElTargetVel := 0;
						bElCtrlBit8 := TRUE;
					ELSE
						bElCtrlBit8 := FALSE;
					END_IF
				END_IF

			// ----- 模式 5: 待机（停止运动，保持上电）-----
			MODES.halt://待机
				IF NOT sStatus.Disabled THEN
					IF sStatus.Moving THEN
						GVL.diElTargetVel := 0;
						bElCtrlBit8 := TRUE;
					ELSE
						bElCtrlBit8 := FALSE;
					END_IF
				END_IF
			
		END_CASE

	// =========== 本控分支（bLocalCtrl=TRUE）===========
	ELSE // 本控
		IF sLocal.iMode <> 1 THEN
			istate:=0;
			icount:=0;
		END_IF
		CASE sLocal.iMode OF

			MODES.powerOff: // 下电
				IF NOT sStatus.Disabled THEN
					IF sStatus.Moving THEN // 运动中，先停止运动
						GVL.diElTargetVel := 0;
						bElCtrlBit8 := TRUE;
					ELSE
						// 写入下电控制字
						GVL.bElCtrlBit3 := FALSE;
						GVL.bElCtrlBit0 := FALSE;
						GVL.bElCtrlBit1 := FALSE;
						GVL.bElCtrlBit2 := FALSE;
					END_IF
				END_IF

			MODES.powerOn:  // 上电（与远控相同的三步序列）
				IF sStatus.Disabled THEN
					GVL.diElTargetVel := 0;
					IF GVL.siElMode <> 3 THEN // 上电时模式默认为3，速度模式
						GVL.siElMode := 3;
					END_IF
					IF siElMode = 3 THEN
						CASE istate OF
							0:
								GVL.bElCtrlBit1 := TRUE;
								GVL.bElCtrlBit2 := TRUE;
								icount := icount + 1;
								IF icount = 20 THEN
									icount:=0;
									istate:=1;
								END_IF
							1:
								GVL.bElCtrlBit0 := TRUE;
								icount := icount + 1;
								IF icount = 20 THEN
									icount:=0;
									istate:=2;
								END_IF
							2:
								GVL.bElCtrlBit3 := TRUE;
						END_CASE
					END_IF
				ELSE
					IF sStatus.Moving THEN
						GVL.diElTargetVel := 0;
						bElCtrlBit8 := TRUE;
					ELSE
						bElCtrlBit8 := FALSE;
					END_IF
				END_IF

			MODES.velocityMode://手控速度模式-本控模式
				IF NOT sStatus.Disabled THEN
					IF ABS(sLocal.rVelCmd) <= sLocal.rVel_Limit THEN
						GVL.diElTargetVel := REAL_TO_DINT(sLocal.rVelCmd * 524288 / 360);
					ELSIF sLocal.rVelCmd > sLocal.rVel_Limit THEN
						GVL.diElTargetVel := REAL_TO_DINT(sLocal.rVel_Limit * 524288 / 360);
					ELSE
						GVL.diElTargetVel := REAL_TO_DINT(-sLocal.rVel_Limit * 524288 / 360);
					END_IF
					GVL.diElTargetAcc := REAL_TO_UDINT(sLocal.rAcceleration * 524288 / 360);   //加速度
					GVL.diElTargetDec := REAL_TO_UDINT(sLocal.rDeceleration * 524288 / 360);   //减速度
				END_IF

			MODES.programBootMode://本控位置模式（普通 PID，不用变增益）
				IF NOT sStatus.Disabled THEN
					IF NOT sLocal.bPIDEnable THEN
						GVL.diElTargetVel := 0;							
					ELSE
						IF NOT slocal.bStartAutoTrack THEN
							// 纯位置跟踪 PID
							 VelPID_2(rTarget:=sLocal.rPosCmd,
									 rFeedback:=rRealPos,
									 rPosLimPositive:=sLocal.rSoft_limit_Postive,//软限位
									 rPosLimNegative:=sLocal.rSoft_limit_Negative,
									 rKp:=0.7,
									 rKi:=0,
									 rKd:=0,
									 iThreshold:=sLocal.rPIDThre,
									 bPIDEnable:=sLocal.bPIDEnable,
									 rVelLim:=sLocal.Pos_Vel,
									 rPIDOutput=>sLocal.rPIDCmdVel);//普通PID
						ELSE
							// 本控自跟踪：误差电压叠加
							 VelPID_2(rTarget:=sLocal.rChanU + rRealPos,
								rFeedback:=rRealPos,
								rPosLimPositive:=sLocal.rSoft_limit_Postive,
								rPosLimNegative:=sLocal.rSoft_limit_Negative,
								rVelLim:=sLocal.rVel_Limit,
								rKp:=1,//自跟踪PI系数3,0.02
								rKi:=0,
								rKd:=0,
								bPIDEnable:=sLocal.bPIDEnable,
								iThreshold:= -1,
								rPIDOutput=>sLocal.rPIDCmdVel);
						END_IF
						
					END_IF
					GVL.diElTargetVel := REAL_TO_DINT(sLocal.rPIDCmdVel * 524288 / 360);
					GVL.diElTargetAcc := REAL_TO_UDINT(9 * 524288 / 360);   //加速度
					GVL.diElTargetDec := REAL_TO_UDINT(9 * 524288 / 360);   //减速度
				END_IF

			MODES.reset://重置
			// 是否需要
			MODES.halt://待机
				IF NOT sStatus.Disabled THEN
					IF sStatus.Moving THEN
						GVL.diElTargetVel := 0;
						bElCtrlBit8 := TRUE;
					ELSE
						bElCtrlBit8 := FALSE;
					END_IF
				END_IF
			
		END_CASE
	END_IF

// =============================================================================
// 段 E: 全局错误时强制停轴（Error_code≠0 但驱动本身无错，属于上层逻辑错误）
// 发快速停止，超时 1s 后强制下电
// =============================================================================
ELSIF GVL.Error_code<>0 AND GVL.eElErrorcode = 0 AND NOT GVL.bElCtrlBit7  AND NOT tr AND NOT bfin1 AND NOT bfin2 THEN
	// 出现错误，轴停止运动
	GVL.diElTargetVel := 0;
	bElCtrlBit8 := TRUE;
	TON_0(IN:=bElCtrlBit8,PT:=T#1S,Q=>,ET=>);//判断stop0执行是否超时,若超时强制下电（手动复位）
	IF TON_0.Q THEN
		bTick:=TRUE;
	END_IF
	IF bTick AND sStatus.Moving THEN // 超时强制下电
		// 写入下电控制字
		GVL.bElCtrlBit3 := FALSE;
		GVL.bElCtrlBit0 := FALSE;
		GVL.bElCtrlBit1 := FALSE;
		GVL.bElCtrlBit2 := FALSE;
	END_IF
END_IF

                  
END_FUNCTION_BLOCK

PROGRAM El_ctrl_1
  VAR
    Axis1_Ctrl : El_Ctrl_FB;  (* 俯仰轴控制 FB（阶段 4 已注释） *)
    bRemote2LocalStop : BOOL;  (* 远控→本控切换中，需先减速下电 *)
    bLocal2RemoteStop : BOOL;  (* 本控→远控切换中，需先减速下电 *)
    Error : INT;  (* 保留 *)
    Axis1Limit_pos : REAL;  (* 硬限位上限 180° *)
    Axis1Limit_Neg : REAL;  (* 硬限位下限 93° *)
    bRTriger : Standard.R_TRIG;  (* bLocalCtrl 上升沿（切到本控） *)
    bFTriger : Standard.F_TRIG;  (* bLocalCtrl 下降沿（切到远控） *)
    Stop1_Count : INT;  (* 低速持续计数（用于判定已停稳） *)
    bStop_1 : BOOL;  (* TRUE=俯仰轴已停稳（|v|<0.035 持续>1s） *)
    rPosModeStepBias : LREAL;  (* 保留/指向模式步进偏置 *)
    rPosModeStep : LREAL;
    rStepBiasMax : LREAL;
    rStepBias : LREAL;  (* Modbus 下发的手动偏置，逐步逼近 rBias_1 *)
    rStep : LREAL;  (* rStepBias 每拍变化步长 *)
    rAuToStepBias : LREAL;  (* 自跟踪累积拉偏 (deg) *)
    rAuToStepBiasTemp : LREAL;  (* 自跟踪瞬时拉偏分量 *)
    rAutoStep : LREAL;  (* 关闭自跟踪后 rAuToStepBias 归零步长 *)
    TbAutoTrigger : Standard.F_TRIG;
    RbAutoTrigger : Standard.R_TRIG;
    rAutoTrackingBiasMax : LREAL;  (* 自跟踪拉偏上限 *)
    rLocalInitPosModeSpeed : REAL;
    rRemoteInitPosModeSpeed : REAL;
    iCountOffAuto : INT;
    iCasePBAutoTrack : INT;
    rKAuToStepBias : LREAL;  (* 自跟踪拉偏增益系数 *)
    agcmaxsearch_tb : AGCMaxSearch_PB_1;  (* 指向模式(mode2) AGC 峰值搜索 *)
    rSearchNextStepTarget_tb : REAL;  (* 指向模式搜索输出偏置 *)
    agcmaxsearch_pb : AGCMaxSearch_PB_1;  (* 程引模式(mode4) AGC 峰值搜索 *)
    rElthreshold : REAL;  (* 俯仰角阈值：仅高于此值才在程引下做 AGC 搜索 *)
    toN1 : Standard.Ton;
    ttime1 : TIME;
    bstartagcmaxsearch : BOOL;
    rSearchNextStepTarget : REAL;  (* 程引模式 AGC 搜索输出偏置 *)
    rMaxPosTest : REAL;  (* AGC 搜索调试：峰值位置 *)
  END_VAR

                    
(*==============================================================================
  PRG: El_ctrl_1（俯仰轴 El 顶层程序）
  任务: Canopen 10ms
  作用:
    1. 读 CANopen 反馈 → 换算实际速度/位置 (rFctVelReal_1 / rFctPosReal_1)
    2. 组装 Axis1Status（故障、使能、运动中等）
    3. 远/本控切换保护、自跟踪拉偏、AGC 峰值搜索
    4. 合成 PID 目标位置 rPIDCmdPos → 调用 El_Ctrl_FB
  数据流:
    Modbus/上位机 → Axis1Remote（在 Modbus_Slave 等处赋值）
    RealTimePosCal.rInterElPos + 各类偏置 → rPIDCmdPos → El_Ctrl_FB → GVL.diEl*
==============================================================================*)




(* 远控参量曾在此从 Modbus_Slave 直赋，现改由 Modbus_Slave 程序统一写入 Axis1Remote *)

// =============================================================================
// 段 1: 驱动状态字 → Axis1Status（供 El_Ctrl_FB 与 HMI 使用）
// DS402 状态: bit0/1/2 同时为 1 表示 Operation Enabled（伺服已使能）
// =============================================================================
Axis1Status.Error := GVL.bElStsBit3;
Axis1Status.ErrorID := GVL.eElErrorcode;
Axis1Status.bServo_Enable := GVL.bElStsBit0 AND GVL.bElStsBit1 AND GVL.bElStsBit2;
Axis1Status.bBrake := NOT (GVL.bElStsBit0 AND GVL.bElStsBit1 AND GVL.bElStsBit2);
Axis1Status.Disabled := NOT (GVL.bElStsBit0 AND GVL.bElStsBit1 AND GVL.bElStsBit2);
// 软限位写入命令结构体（与下面硬限位 93~180 一致）
Axis1Remote.rSoft_limit_Negative:=93;Axis1Remote.rSoft_limit_Postive:=180;
Axis1Local.rSoft_limit_Negative:=93;Axis1Local.rSoft_limit_Postive:=180;

// =============================================================================
// 段 2: CANopen 反馈 → 实际速度/位置（deg, deg/s）
// 公式: 物理量 = diActXxx / 524288 × 360；俯仰另加 Modbus 标定偏移 lrElOffset
// =============================================================================
rFctVelReal_1:=DINT_TO_REAL(diElActVel)/524288.0*360.0;
rFctPosReal_1:=DINT_TO_REAL(diElActPos)/524288.0*360.0 + modbus_slave.lrElOffset;

// =============================================================================
// 段 3: 指向命令硬限位（远控/本控 rPosCmd 钳位到 93°~180°）
// =============================================================================
Axis1Limit_pos:=180;
Axis1Limit_Neg:=93;
IF Axis1Remote.rPosCmd>Axis1Limit_pos THEN
	Axis1Remote.rPosCmd:=180;
ELSIF Axis1Remote.rPosCmd<Axis1Limit_Neg THEN
	 Axis1Remote.rPosCmd:=93;  
END_IF

IF Axis1Local.rPosCmd>Axis1Limit_pos THEN
	Axis1Local.rPosCmd:=180;
ELSIF Axis1Local.rPosCmd<Axis1Limit_Neg THEN
	 Axis1Local.rPosCmd:=93;  
END_IF

// =============================================================================
// 段 4: 停稳判定 → Axis1Status.Moving
// |速度|<0.035°/s 连续 100 拍(约1s) 认为停稳；bStop_1=TRUE → Moving=FALSE
// =============================================================================
IF  ABS(rFctVelReal_1)<0.035 THEN
	Stop1_Count:=Stop1_Count+1;
	IF Stop1_Count>100 THEN
		Stop1_Count:=101;
		bStop_1:=TRUE;;
	END_IF
ELSE
	Stop1_Count:=0;
	bStop_1:=FALSE;
END_IF
Axis1Status.Moving := NOT bStop_1;

// =============================================================================
// 段 5: PID 使能 — 仅指向(2)与程引(4)模式需要位置环
// =============================================================================
IF Axis1Remote.iMode=2 OR Axis1Remote.iMode=4 THEN
	Axis1Remote.bPIDEnable:=TRUE;
ELSE
	Axis1Remote.bPIDEnable:=FALSE;
END_IF

// =============================================================================
// 段 6: 远控 ↔ 本控 切换保护（GVL.bLocalCtrl）
// 切换瞬间若伺服仍使能 → 置切换标志 → 强制 mode=7(halt) 减速
// 停稳且下电完成后 → mode=0，清除标志
// =============================================================================
bRTriger(CLK:=GVL.bLocalCtrl);
bFTriger(CLK:=GVL.bLocalCtrl);

// 远控 → 本控（bLocalCtrl 上升沿）
IF Axis1Status.bServo_Enable AND (bRTriger.Q ) THEN//如果速度不为0且本控发生切换，则减速停止标识为True
	bRemote2LocalStop:=TRUE;
END_IF
IF bRemote2LocalStop  THEN //若减速停止标识符为True 
	
	IF  bStop_1=TRUE THEN//且电机速度不为0 开始减速 减速完成后下使能，下使能完成后复位标识符复位
		Axis1Local.iMode:=0;
		Axis1Remote.iMode:=0;
		IF Axis1Status.bServo_Enable=FALSE THEN
			bRemote2LocalStop:=FALSE;
		END_IF
	ELSE
		Axis1Local.iMode:=7;
		Axis1Remote.iMode:=7;
	END_IF
END_IF

// 本控 → 远控（bLocalCtrl 下降沿）
IF Axis1Status.bServo_Enable AND (bFTriger.Q ) THEN//如果速度不为0且本控发生切换，则减速停止标识为True
	bLocal2RemoteStop:=TRUE;
END_IF
IF bLocal2RemoteStop  THEN //若减速停止标识符为True 
	
	IF  bStop_1=TRUE THEN//且电机速度不为0 开始减速 减速完成后下使能，下使能完成后复位标识符复位
		Axis1Local.iMode:=0;
		Axis1Remote.iMode:=0;
		IF Axis1Status.bServo_Enable=FALSE THEN
			bLocal2RemoteStop:=FALSE;
		END_IF
	ELSE
		Axis1Remote.iMode:=7;
		Axis1Local.iMode:=7;
	END_IF
END_IF

// =============================================================================
// 段 7: AGC 峰值搜索（与方位 Az_ctrl_1 协同，bstartSearchEl 由方位触发）
// mode2: 插值目标 = rPosCmd；mode4: 插值目标 = RealTimePosCal.rInterElPos
// 仅当俯仰高于 rElthreshold（相对水平）且在程引下才在 mode4 启用搜索
// =============================================================================
IF Axis1Remote.iMode=2 THEN
			IF GVL.Chan1AGC>=(GVL.Chanthreshold-0.1) THEN
					agcmaxsearch_pb(bstart:=Az_ctrl_1.agcmaxsearch_tb.bSucess,rAGCNow:=GVL.Chan1AGC,btrig:=Az_ctrl_1.bstartSearchEl,
						rCurrentPos:=rFctPosReal_1,rInterPos:=Axis1Remote.rPosCmd,
				rStepBiasNow:=rStepBias,bAutoTracking:=GVL.bStartTrack,bStop:=FALSE,
				rStepBias=>rSearchNextStepTarget_tb,rAGCMaxBias=>rMaxPosTest,bSucess=>);
			ELSE
				bstartagcmaxsearch:=FALSE;
				agcmaxsearch_pb(bstart:=Az_ctrl_1.agcmaxsearch_tb.bSucess,rAGCNow:=GVL.Chan1AGC,btrig:=Az_ctrl_1.bstartSearchEl,
				rCurrentPos:=rFctPosReal_1,rInterPos:=Axis1Remote.rPosCmd,
				rStepBiasNow:=rStepBias,bAutoTracking:=GVL.bStartTrack,bStop:=FALSE,
				rStepBias=>rSearchNextStepTarget_tb,rAGCMaxBias=>rMaxPosTest,bSucess=>);
			END_IF
		ELSIF Axis1Remote.iMode=4 AND rFctPosReal_1-90>rElthreshold  THEN
			IF GVL.Chan1AGC>=(GVL.Chanthreshold-0.1) THEN
					agcmaxsearch_pb(bstart:=Az_ctrl_1.agcmaxsearch_pb.bSucess,rAGCNow:=GVL.Chan1AGC,btrig:=Az_ctrl_1.bstartSearchEl,
						rCurrentPos:=rFctPosReal_1,rInterPos:=RealTimePosCal.rInterElPos,
				rStepBiasNow:=rStepBias,bAutoTracking:=GVL.bStartTrack,bStop:=FALSE,
				rStepBias=>rSearchNextStepTarget,rAGCMaxBias=>rMaxPosTest,bSucess=>);
			ELSE
				bstartagcmaxsearch:=FALSE;
				agcmaxsearch_pb(bstart:=Az_ctrl_1.agcmaxsearch_pb.bSucess,rAGCNow:=GVL.Chan1AGC,btrig:=Az_ctrl_1.bstartSearchEl,
				rCurrentPos:=rFctPosReal_1,rInterPos:=RealTimePosCal.rInterElPos,
				rStepBiasNow:=rStepBias,bAutoTracking:=GVL.bStartTrack,bStop:=FALSE,
				rStepBias=>rSearchNextStepTarget,rAGCMaxBias=>rMaxPosTest,bSucess=>);
			END_IF
		ELSIF Axis1Remote.iMode =0  OR Axis1Remote.iMode =7 THEN
			bstartagcmaxsearch:=FALSE;
			agcmaxsearch_pb(bstart:=Az_ctrl_1.agcmaxsearch_pb.bSucess,rAGCNow:=GVL.Chan1AGC,btrig:=Az_ctrl_1.bstartSearchEl,
			rCurrentPos:=rFctPosReal_1,rInterPos:=RealTimePosCal.rInterElPos,	
			rStepBiasNow:=rStepBias,bAutoTracking:=GVL.bStartTrack,bStop:=FALSE,
			rStepBias=>rSearchNextStepTarget,rAGCMaxBias=>rMaxPosTest,bSucess=>);
		END_IF

// =============================================================================
// 段 8: 自跟踪拉偏（远控）
// mode4+程引: 用 AutoTrackingCal.rChanUe 累积 rAuToStepBias（限幅）
// mode2+指向: 直接用 rChanU 作 PID 目标增量（在 El_Ctrl_FB 内 rChanU+位置）
// 关跟踪: rAuToStepBias 渐零，rStepBias 渐近 Modbus_Slave.rBias_1
// =============================================================================
IF GVL.bStartTrack AND Axis1Remote.iMode=4 THEN
	Axis1Remote.bStartAutoTrack := TRUE;
	IF rAuToStepBias > rAutoTrackingBiasMax THEN
		rAuToStepBias := rAutoTrackingBiasMax;
	ELSIF rAuToStepBias < -rAutoTrackingBiasMax THEN
		rAuToStepBias := -rAutoTrackingBiasMax;
	ELSE
		rAuToStepBiasTemp:=0.02*AutoTrackingCal.rDirSenFac*AutoTrackingCal.rChanUe;
		rAuToStepBias:=rAuToStepBias+AutoTrackingCal.rDirSenFac*rKAuToStepBias*AutoTrackingCal.rChanUe/1000.0;
	END_IF
ELSIF NOT GVL.bStartTrack AND Axis1Remote.iMode=4 THEN
	IF 	rAuToStepBias>0 THEN//关闭自跟踪后自跟踪拉偏量逐渐归0
		rAuToStepBias:=rAuToStepBias-rAutoStep;
	ELSIF rAuToStepBias<0 THEN
		rAuToStepBias:=rAuToStepBias+rAutoStep;
	ELSE
		rAuToStepBias:=0;
	END_IF
	
	IF Modbus_Slave.rBias_1>rStepBias THEN
		rStepBias:=rStepBias+rStep;
		IF rStepBias>=Modbus_Slave.rBias_1 THEN
			rStepBias:=Modbus_Slave.rBias_1;
		END_IF
	ELSIF Modbus_Slave.rBias_1<rStepBias THEN
		rStepBias:=rStepBias-rStep;
		IF rStepBias<=Modbus_Slave.rBias_1 THEN
			rStepBias:=Modbus_Slave.rBias_1;
		END_IF
	END_IF
	rAuToStepBiasTemp:=0;
ELSIF GVL.bStartTrack AND Axis1Remote.iMode=2 THEN
	Axis1Remote.bStartAutoTrack := TRUE;
	Axis1Remote.rChanU := AutoTrackingCal.rChanUe;
ELSE
	Axis1Remote.bStartAutoTrack := FALSE;	
	rAuToStepBias:=0;
	rStepBias:=0;
	rAuToStepBiasTemp:=0;
END_IF

// 本控自跟踪（仅程引 mode4）
IF GVL.bStartLocalAutoTrack AND Axis1Local.iMode = 4 THEN
	Axis1Local.bStartAutoTrack := TRUE;
	Axis1Local.rChanU := AutoTrackingCal.rChanUeLocal;
ELSE
	Axis1Local.bStartAutoTrack := FALSE;
END_IF

